      movel([0.335259, -1.470222, -2.504094, -0.738074, 1.570796, 1.906055],accel_mss,speed_ms,0,blend_radius_m)
      movel([0.336291, -1.468662, -2.505402, -0.738325, 1.570796, 1.907087],accel_mss,speed_ms,0,blend_radius_m)
      movel([0.337329, -1.467098, -2.506710, -0.738581, 1.570796, 1.908125],accel_mss,speed_ms,0,blend_radius_m)
      movel([0.339195, -1.464306, -2.509036, -0.739047, 1.570796, 1.909991],accel_mss,speed_ms,0,blend_radius_m)
      movel([0.339233, -1.464257, -2.509076, -0.739055, 1.570796, 1.910029],accel_mss,speed_ms,0,blend_radius_m)
      movel([0.339275, -1.464212, -2.509113, -0.739063, 1.570796, 1.910071],accel_mss,speed_ms,0,blend_radius_m)
      movel([0.339324, -1.464171, -2.509148, -0.739070, 1.570796, 1.910121],accel_mss,speed_ms,0,blend_radius_m)
      movel([0.339395, -1.464123, -2.509187, -0.739078, 1.570796, 1.910192],accel_mss,speed_ms,0,blend_radius_m)
      movel([0.339472, -1.464083, -2.509221, -0.739085, 1.570796, 1.910268],accel_mss,speed_ms,0,blend_radius_m)
      movel([0.339550, -1.464051, -2.509248, -0.739090, 1.570796, 1.910346],accel_mss,speed_ms,0,blend_radius_m)
      movel([0.339628, -1.464028, -2.509266, -0.739094, 1.570796, 1.910425],accel_mss,speed_ms,0,blend_radius_m)
      movel([0.343643, -1.463141, -2.510002, -0.739245, 1.570796, 1.914440],accel_mss,speed_ms,0,blend_radius_m)
      movel([0.345543, -1.462730, -2.510343, -0.739316, 1.570796, 1.916340],accel_mss,speed_ms,0,blend_radius_m)
      movel([0.347442, -1.462325, -2.510678, -0.739385, 1.570796, 1.918239],accel_mss,speed_ms,0,blend_radius_m)
      movel([0.347658, -1.462283, -2.510713, -0.739393, 1.570796, 1.918454],accel_mss,speed_ms,0,blend_radius_m)
      movel([0.347869, -1.462252, -2.510739, -0.739398, 1.570796, 1.918666],accel_mss,speed_ms,0,blend_radius_m)
      movel([0.348080, -1.462228, -2.510759, -0.739402, 1.570796, 1.918876],accel_mss,speed_ms,0,blend_radius_m)
      movel([0.348287, -1.462214, -2.510770, -0.739405, 1.570796, 1.919083],accel_mss,speed_ms,0,blend_radius_m)
      movel([0.348391, -1.462213, -2.510771, -0.739405, 1.570796, 1.919187],accel_mss,speed_ms,0,blend_radius_m)
      movel([0.348491, -1.462224, -2.510762, -0.739403, 1.570796, 1.919287],accel_mss,speed_ms,0,blend_radius_m)
      movel([0.348582, -1.462246, -2.510744, -0.739399, 1.570796, 1.919378],accel_mss,speed_ms,0,blend_radius_m)
      movel([0.348667, -1.462277, -2.510718, -0.739394, 1.570796, 1.919464],accel_mss,speed_ms,0,blend_radius_m)
      movel([0.355079, -1.465147, -2.508336, -0.738906, 1.570796, 1.925875],accel_mss,speed_ms,0,blend_radius_m)
      movel([0.361512, -1.468104, -2.505869, -0.738416, 1.570796, 1.932309],accel_mss,speed_ms,0,blend_radius_m)
      speed_ms = 0.003
      movel([0.361512, -1.456047, -2.500408, -0.755934, 1.570796, 1.932309],accel_mss,speed_ms,0,blend_radius_m)
      speed_ms = 0.01
      movel([0.361512, -1.432785, -2.489096, -0.790508, 1.570796, 1.932309],accel_mss,speed_ms,0,blend_radius_m)
      movel([0.379710, -1.378240, -2.530192, -0.803957, 1.570796, 1.950507],accel_mss,speed_ms,0,blend_radius_m)
      movel([0.379710, -1.402570, -2.542172, -0.767647, 1.570796, 1.950507],accel_mss,speed_ms,0,blend_radius_m)
      speed_ms = 0.003
      movel([0.379710, -1.412031, -2.546529, -0.753828, 1.570796, 1.950507],accel_mss,speed_ms,0,blend_radius_m)
      speed_ms = 0.007
      movel([0.362253, -1.410756, -2.547488, -0.754145, 1.570796, 1.933049],accel_mss,speed_ms,0,blend_radius_m)
      movel([0.344648, -1.409792, -2.548210, -0.754386, 1.570796, 1.915445],accel_mss,speed_ms,0,blend_radius_m)
      movel([0.344585, -1.409783, -2.548217, -0.754389, 1.570796, 1.915381],accel_mss,speed_ms,0,blend_radius_m)
      movel([0.344531, -1.409760, -2.548234, -0.754395, 1.570796, 1.915327],accel_mss,speed_ms,0,blend_radius_m)
      movel([0.344488, -1.409724, -2.548261, -0.754404, 1.570796, 1.915285],accel_mss,speed_ms,0,blend_radius_m)
      movel([0.344479, -1.409701, -2.548278, -0.754409, 1.570796, 1.915276],accel_mss,speed_ms,0,blend_radius_m)
      movel([0.344486, -1.409671, -2.548301, -0.754417, 1.570796, 1.915282],accel_mss,speed_ms,0,blend_radius_m)
      movel([0.345097, -1.408321, -2.549311, -0.754757, 1.570796, 1.915893],accel_mss,speed_ms,0,blend_radius_m)
      movel([0.345789, -1.406806, -2.550440, -0.755143, 1.570796, 1.916585],accel_mss,speed_ms,0,blend_radius_m)
      movel([0.346623, -1.405010, -2.551775, -0.755604, 1.570796, 1.917420],accel_mss,speed_ms,0,blend_radius_m)
      movel([0.348821, -1.400311, -2.555246, -0.756833, 1.570796, 1.919617],accel_mss,speed_ms,0,blend_radius_m)
      movel([0.349537, -1.400351, -2.555216, -0.756822, 1.570796, 1.920333],accel_mss,speed_ms,0,blend_radius_m)
      movel([0.355122, -1.400638, -2.555005, -0.756746, 1.570796, 1.925918],accel_mss,speed_ms,0,blend_radius_m)
      movel([0.367492, -1.401377, -2.554461, -0.756551, 1.570796, 1.938288],accel_mss,speed_ms,0,blend_radius_m)
      movel([0.384563, -1.402661, -2.553514, -0.756214, 1.570796, 1.955359],accel_mss,speed_ms,0,blend_radius_m)
      movel([0.384371, -1.403120, -2.553175, -0.756094, 1.570796, 1.955168],accel_mss,speed_ms,0,blend_radius_m)
      movel([0.384269, -1.403350, -2.553005, -0.756034, 1.570796, 1.955065],accel_mss,speed_ms,0,blend_radius_m)
      movel([0.384107, -1.403677, -2.552763, -0.755949, 1.570796, 1.954904],accel_mss,speed_ms,0,blend_radius_m)
      movel([0.383922, -1.404034, -2.552499, -0.755856, 1.570796, 1.954719],accel_mss,speed_ms,0,blend_radius_m)
      movel([0.383739, -1.404372, -2.552248, -0.755769, 1.570796, 1.954535],accel_mss,speed_ms,0,blend_radius_m)
      movel([0.383297, -1.405163, -2.551661, -0.755564, 1.570796, 1.954093],accel_mss,speed_ms,0,blend_radius_m)
      movel([0.381035, -1.405216, -2.551623, -0.755551, 1.570796, 1.951831],accel_mss,speed_ms,0,blend_radius_m)
      movel([0.378702, -1.405326, -2.551541, -0.755522, 1.570796, 1.949498],accel_mss,speed_ms,0,blend_radius_m)
      movel([0.378649, -1.405401, -2.551485, -0.755503, 1.570796, 1.949445],accel_mss,speed_ms,0,blend_radius_m)
      movel([0.377743, -1.408698, -2.549029, -0.754662, 1.570796, 1.948539],accel_mss,speed_ms,0,blend_radius_m)
      movel([0.381641, -1.408475, -2.549196, -0.754719, 1.570796, 1.952437],accel_mss,speed_ms,0,blend_radius_m)
      movel([0.380797, -1.410194, -2.547909, -0.754286, 1.570796, 1.951594],accel_mss,speed_ms,0,blend_radius_m)
      movel([0.380468, -1.410858, -2.547411, -0.754120, 1.570796, 1.951265],accel_mss,speed_ms,0,blend_radius_m)
      movel([0.380174, -1.411429, -2.546983, -0.753978, 1.570796, 1.950970],accel_mss,speed_ms,0,blend_radius_m)
      movel([0.379918, -1.411918, -2.546614, -0.753856, 1.570796, 1.950714],accel_mss,speed_ms,0,blend_radius_m)
      movel([0.379892, -1.411953, -2.546588, -0.753848, 1.570796, 1.950688],accel_mss,speed_ms,0,blend_radius_m)
      movel([0.379860, -1.411982, -2.546567, -0.753841, 1.570796, 1.950656],accel_mss,speed_ms,0,blend_radius_m)
      movel([0.379809, -1.412013, -2.546544, -0.753833, 1.570796, 1.950606],accel_mss,speed_ms,0,blend_radius_m)
      movel([0.379758, -1.412028, -2.546532, -0.753829, 1.570796, 1.950555],accel_mss,speed_ms,0,blend_radius_m)
      movel([0.379710, -1.412031, -2.546529, -0.753828, 1.570796, 1.950507],accel_mss,speed_ms,0,blend_radius_m)
      speed_ms = 0.003
      movel([0.379710, -1.415226, -2.547965, -0.749197, 1.570796, 1.950507],accel_mss,speed_ms,0,blend_radius_m)
      speed_ms = 0.007
      movel([0.362253, -1.413954, -2.548926, -0.749509, 1.570796, 1.933049],accel_mss,speed_ms,0,blend_radius_m)
      movel([0.344648, -1.412994, -2.549649, -0.749746, 1.570796, 1.915445],accel_mss,speed_ms,0,blend_radius_m)
      movel([0.344585, -1.412984, -2.549657, -0.749748, 1.570796, 1.915381],accel_mss,speed_ms,0,blend_radius_m)
      movel([0.344531, -1.412962, -2.549674, -0.749754, 1.570796, 1.915327],accel_mss,speed_ms,0,blend_radius_m)
      movel([0.344488, -1.412926, -2.549701, -0.749763, 1.570796, 1.915285],accel_mss,speed_ms,0,blend_radius_m)
      movel([0.344479, -1.412903, -2.549718, -0.749768, 1.570796, 1.915276],accel_mss,speed_ms,0,blend_radius_m)
      movel([0.344486, -1.412873, -2.549740, -0.749776, 1.570796, 1.915282],accel_mss,speed_ms,0,blend_radius_m)
      movel([0.345097, -1.411526, -2.550752, -0.750110, 1.570796, 1.915893],accel_mss,speed_ms,0,blend_radius_m)
      movel([0.345789, -1.410016, -2.551885, -0.750489, 1.570796, 1.916585],accel_mss,speed_ms,0,blend_radius_m)
      movel([0.346623, -1.408225, -2.553222, -0.750942, 1.570796, 1.917420],accel_mss,speed_ms,0,blend_radius_m)
      movel([0.348821, -1.403539, -2.556700, -0.752150, 1.570796, 1.919617],accel_mss,speed_ms,0,blend_radius_m)
      movel([0.349537, -1.403579, -2.556670, -0.752139, 1.570796, 1.920333],accel_mss,speed_ms,0,blend_radius_m)
      movel([0.355122, -1.403865, -2.556459, -0.752065, 1.570796, 1.925918],accel_mss,speed_ms,0,blend_radius_m)
      movel([0.367492, -1.404602, -2.555914, -0.751873, 1.570796, 1.938288],accel_mss,speed_ms,0,blend_radius_m)
      movel([0.384563, -1.405883, -2.554965, -0.751542, 1.570796, 1.955359],accel_mss,speed_ms,0,blend_radius_m)
      movel([0.384371, -1.406340, -2.554625, -0.751424, 1.570796, 1.955168],accel_mss,speed_ms,0,blend_radius_m)
      movel([0.384269, -1.406569, -2.554455, -0.751365, 1.570796, 1.955065],accel_mss,speed_ms,0,blend_radius_m)
      movel([0.384107, -1.406895, -2.554212, -0.751281, 1.570796, 1.954904],accel_mss,speed_ms,0,blend_radius_m)
      movel([0.383922, -1.407252, -2.553947, -0.751190, 1.570796, 1.954719],accel_mss,speed_ms,0,blend_radius_m)
      movel([0.383739, -1.407589, -2.553696, -0.751104, 1.570796, 1.954535],accel_mss,speed_ms,0,blend_radius_m)
      movel([0.383297, -1.408378, -2.553108, -0.750903, 1.570796, 1.954093],accel_mss,speed_ms,0,blend_radius_m)
      movel([0.381035, -1.408430, -2.553069, -0.750890, 1.570796, 1.951831],accel_mss,speed_ms,0,blend_radius_m)
      movel([0.378702, -1.408540, -2.552987, -0.750862, 1.570796, 1.949498],accel_mss,speed_ms,0,blend_radius_m)
      movel([0.378649, -1.408615, -2.552931, -0.750843, 1.570796, 1.949445],accel_mss,speed_ms,0,blend_radius_m)
      movel([0.377743, -1.411903, -2.550470, -0.750016, 1.570796, 1.948539],accel_mss,speed_ms,0,blend_radius_m)
      movel([0.381641, -1.411680, -2.550637, -0.750072, 1.570796, 1.952437],accel_mss,speed_ms,0,blend_radius_m)
      movel([0.380797, -1.413394, -2.549348, -0.749647, 1.570796, 1.951594],accel_mss,speed_ms,0,blend_radius_m)
      movel([0.380468, -1.414056, -2.548849, -0.749484, 1.570796, 1.951265],accel_mss,speed_ms,0,blend_radius_m)
      movel([0.380174, -1.414625, -2.548419, -0.749344, 1.570796, 1.950970],accel_mss,speed_ms,0,blend_radius_m)
      movel([0.379918, -1.415114, -2.548050, -0.749225, 1.570796, 1.950714],accel_mss,speed_ms,0,blend_radius_m)
      movel([0.379892, -1.415148, -2.548024, -0.749217, 1.570796, 1.950688],accel_mss,speed_ms,0,blend_radius_m)
      movel([0.379860, -1.415177, -2.548003, -0.749210, 1.570796, 1.950656],accel_mss,speed_ms,0,blend_radius_m)
      movel([0.379809, -1.415208, -2.547979, -0.749202, 1.570796, 1.950606],accel_mss,speed_ms,0,blend_radius_m)
      movel([0.379758, -1.415223, -2.547967, -0.749198, 1.570796, 1.950555],accel_mss,speed_ms,0,blend_radius_m)
      movel([0.379710, -1.415226, -2.547965, -0.749197, 1.570796, 1.950507],accel_mss,speed_ms,0,blend_radius_m)
      speed_ms = 0.003
      movel([0.379710, -1.402570, -2.542172, -0.767647, 1.570796, 1.950507],accel_mss,speed_ms,0,blend_radius_m)
      speed_ms = 0.01
      movel([0.379710, -1.378240, -2.530192, -0.803957, 1.570796, 1.950507],accel_mss,speed_ms,0,blend_radius_m)
      movel([0.382022, -1.366015, -2.538831, -0.807543, 1.570796, 1.952818],accel_mss,speed_ms,0,blend_radius_m)
      movel([0.382022, -1.390572, -2.550964, -0.770853, 1.570796, 1.952818],accel_mss,speed_ms,0,blend_radius_m)
      speed_ms = 0.003
      movel([0.382022, -1.400129, -2.555379, -0.756881, 1.570796, 1.952818],accel_mss,speed_ms,0,blend_radius_m)
      speed_ms = 0.007
      movel([0.381906, -1.400143, -2.555369, -0.756877, 1.570796, 1.952702],accel_mss,speed_ms,0,blend_radius_m)
      movel([0.381797, -1.400145, -2.555368, -0.756877, 1.570796, 1.952593],accel_mss,speed_ms,0,blend_radius_m)
      movel([0.381615, -1.400131, -2.555378, -0.756880, 1.570796, 1.952411],accel_mss,speed_ms,0,blend_radius_m)
      movel([0.381436, -1.400113, -2.555391, -0.756885, 1.570796, 1.952232],accel_mss,speed_ms,0,blend_radius_m)
      movel([0.380003, -1.399974, -2.555493, -0.756922, 1.570796, 1.950799],accel_mss,speed_ms,0,blend_radius_m)
      movel([0.365041, -1.398928, -2.556261, -0.757200, 1.570796, 1.935837],accel_mss,speed_ms,0,blend_radius_m)
      movel([0.349510, -1.398092, -2.556873, -0.757424, 1.570796, 1.920307],accel_mss,speed_ms,0,blend_radius_m)
      movel([0.348976, -1.398094, -2.556871, -0.757423, 1.570796, 1.919772],accel_mss,speed_ms,0,blend_radius_m)
      movel([0.348929, -1.398092, -2.556873, -0.757424, 1.570796, 1.919725],accel_mss,speed_ms,0,blend_radius_m)
      movel([0.348886, -1.398079, -2.556882, -0.757427, 1.570796, 1.919683],accel_mss,speed_ms,0,blend_radius_m)
      movel([0.348854, -1.398057, -2.556898, -0.757433, 1.570796, 1.919650],accel_mss,speed_ms,0,blend_radius_m)
      movel([0.348827, -1.398026, -2.556921, -0.757442, 1.570796, 1.919624],accel_mss,speed_ms,0,blend_radius_m)
      movel([0.348812, -1.397990, -2.556947, -0.757451, 1.570796, 1.919608],accel_mss,speed_ms,0,blend_radius_m)
      movel([0.348808, -1.397947, -2.556979, -0.757463, 1.570796, 1.919604],accel_mss,speed_ms,0,blend_radius_m)
      movel([0.348816, -1.397841, -2.557057, -0.757491, 1.570796, 1.919613],accel_mss,speed_ms,0,blend_radius_m)
      movel([0.348845, -1.397731, -2.557137, -0.757521, 1.570796, 1.919641],accel_mss,speed_ms,0,blend_radius_m)
      movel([0.348908, -1.397546, -2.557272, -0.757571, 1.570796, 1.919705],accel_mss,speed_ms,0,blend_radius_m)
      movel([0.348977, -1.397359, -2.557409, -0.757621, 1.570796, 1.919774],accel_mss,speed_ms,0,blend_radius_m)
      movel([0.349097, -1.397073, -2.557618, -0.757698, 1.570796, 1.919894],accel_mss,speed_ms,0,blend_radius_m)
      movel([0.349227, -1.396787, -2.557827, -0.757775, 1.570796, 1.920023],accel_mss,speed_ms,0,blend_radius_m)
      movel([0.351083, -1.392872, -2.560673, -0.758844, 1.570796, 1.921879],accel_mss,speed_ms,0,blend_radius_m)
      movel([0.353252, -1.388325, -2.563951, -0.760113, 1.570796, 1.924049],accel_mss,speed_ms,0,blend_radius_m)
      movel([0.355797, -1.383031, -2.567730, -0.761628, 1.570796, 1.926593],accel_mss,speed_ms,0,blend_radius_m)
      movel([0.362519, -1.369156, -2.577443, -0.765790, 1.570796, 1.933315],accel_mss,speed_ms,0,blend_radius_m)
      movel([0.363532, -1.369162, -2.577439, -0.765788, 1.570796, 1.934328],accel_mss,speed_ms,0,blend_radius_m)
      movel([0.364039, -1.369170, -2.577434, -0.765786, 1.570796, 1.934835],accel_mss,speed_ms,0,blend_radius_m)
      movel([0.364541, -1.369192, -2.577419, -0.765779, 1.570796, 1.935337],accel_mss,speed_ms,0,blend_radius_m)
      movel([0.365033, -1.369226, -2.577395, -0.765768, 1.570796, 1.935829],accel_mss,speed_ms,0,blend_radius_m)
      movel([0.365522, -1.369271, -2.577364, -0.765754, 1.570796, 1.936319],accel_mss,speed_ms,0,blend_radius_m)
      movel([0.366251, -1.369359, -2.577303, -0.765727, 1.570796, 1.937047],accel_mss,speed_ms,0,blend_radius_m)
      movel([0.366968, -1.369467, -2.577228, -0.765694, 1.570796, 1.937764],accel_mss,speed_ms,0,blend_radius_m)
      movel([0.367676, -1.369589, -2.577144, -0.765656, 1.570796, 1.938472],accel_mss,speed_ms,0,blend_radius_m)
      movel([0.368391, -1.369734, -2.577044, -0.765611, 1.570796, 1.939187],accel_mss,speed_ms,0,blend_radius_m)
      movel([0.369092, -1.369897, -2.576932, -0.765561, 1.570796, 1.939888],accel_mss,speed_ms,0,blend_radius_m)
      movel([0.369784, -1.370076, -2.576808, -0.765506, 1.570796, 1.940580],accel_mss,speed_ms,0,blend_radius_m)
      movel([0.370258, -1.370210, -2.576715, -0.765464, 1.570796, 1.941054],accel_mss,speed_ms,0,blend_radius_m)
      movel([0.370723, -1.370357, -2.576613, -0.765419, 1.570796, 1.941519],accel_mss,speed_ms,0,blend_radius_m)
      movel([0.371180, -1.370516, -2.576503, -0.765370, 1.570796, 1.941977],accel_mss,speed_ms,0,blend_radius_m)
      movel([0.371629, -1.370684, -2.576387, -0.765318, 1.570796, 1.942425],accel_mss,speed_ms,0,blend_radius_m)
      movel([0.372272, -1.370949, -2.576203, -0.765237, 1.570796, 1.943068],accel_mss,speed_ms,0,blend_radius_m)
      movel([0.372898, -1.371228, -2.576010, -0.765151, 1.570796, 1.943695],accel_mss,speed_ms,0,blend_radius_m)
      movel([0.373510, -1.371527, -2.575803, -0.765059, 1.570796, 1.944307],accel_mss,speed_ms,0,blend_radius_m)
      movel([0.374110, -1.371842, -2.575584, -0.764963, 1.570796, 1.944907],accel_mss,speed_ms,0,blend_radius_m)
      movel([0.374692, -1.372172, -2.575355, -0.764862, 1.570796, 1.945489],accel_mss,speed_ms,0,blend_radius_m)
      movel([0.375259, -1.372520, -2.575113, -0.764756, 1.570796, 1.946055],accel_mss,speed_ms,0,blend_radius_m)
      movel([0.375812, -1.372886, -2.574859, -0.764644, 1.570796, 1.946608],accel_mss,speed_ms,0,blend_radius_m)
      movel([0.376347, -1.373266, -2.574595, -0.764529, 1.570796, 1.947143],accel_mss,speed_ms,0,blend_radius_m)
      movel([0.376865, -1.373662, -2.574318, -0.764408, 1.570796, 1.947661],accel_mss,speed_ms,0,blend_radius_m)
      movel([0.377367, -1.374074, -2.574032, -0.764283, 1.570796, 1.948164],accel_mss,speed_ms,0,blend_radius_m)
      movel([0.377848, -1.374497, -2.573737, -0.764155, 1.570796, 1.948645],accel_mss,speed_ms,0,blend_radius_m)
      movel([0.378310, -1.374937, -2.573430, -0.764023, 1.570796, 1.949107],accel_mss,speed_ms,0,blend_radius_m)
      movel([0.378755, -1.375391, -2.573112, -0.763886, 1.570796, 1.949551],accel_mss,speed_ms,0,blend_radius_m)
      movel([0.379183, -1.375859, -2.572785, -0.763745, 1.570796, 1.949979],accel_mss,speed_ms,0,blend_radius_m)
      movel([0.379591, -1.376342, -2.572447, -0.763600, 1.570796, 1.950388],accel_mss,speed_ms,0,blend_radius_m)
      movel([0.379981, -1.376840, -2.572098, -0.763451, 1.570796, 1.950777],accel_mss,speed_ms,0,blend_radius_m)
      movel([0.380354, -1.377351, -2.571739, -0.763298, 1.570796, 1.951150],accel_mss,speed_ms,0,blend_radius_m)
      movel([0.380706, -1.377876, -2.571371, -0.763142, 1.570796, 1.951502],accel_mss,speed_ms,0,blend_radius_m)
      movel([0.381041, -1.378415, -2.570992, -0.762982, 1.570796, 1.951837],accel_mss,speed_ms,0,blend_radius_m)
      movel([0.381356, -1.378965, -2.570605, -0.762819, 1.570796, 1.952153],accel_mss,speed_ms,0,blend_radius_m)
      movel([0.381656, -1.379536, -2.570203, -0.762651, 1.570796, 1.952452],accel_mss,speed_ms,0,blend_radius_m)
      movel([0.381939, -1.380118, -2.569792, -0.762479, 1.570796, 1.952735],accel_mss,speed_ms,0,blend_radius_m)
      movel([0.382200, -1.380714, -2.569371, -0.762304, 1.570796, 1.952996],accel_mss,speed_ms,0,blend_radius_m)
      movel([0.382442, -1.381320, -2.568943, -0.762126, 1.570796, 1.953238],accel_mss,speed_ms,0,blend_radius_m)
      movel([0.382666, -1.381936, -2.568506, -0.761946, 1.570796, 1.953462],accel_mss,speed_ms,0,blend_radius_m)
      movel([0.382868, -1.382564, -2.568061, -0.761764, 1.570796, 1.953664],accel_mss,speed_ms,0,blend_radius_m)
      movel([0.383052, -1.383202, -2.567609, -0.761579, 1.570796, 1.953848],accel_mss,speed_ms,0,blend_radius_m)
      movel([0.383215, -1.383850, -2.567148, -0.761391, 1.570796, 1.954011],accel_mss,speed_ms,0,blend_radius_m)
      movel([0.383358, -1.384508, -2.566680, -0.761201, 1.570796, 1.954154],accel_mss,speed_ms,0,blend_radius_m)
      movel([0.383483, -1.385174, -2.566205, -0.761010, 1.570796, 1.954279],accel_mss,speed_ms,0,blend_radius_m)
      movel([0.383590, -1.385871, -2.565708, -0.760810, 1.570796, 1.954386],accel_mss,speed_ms,0,blend_radius_m)
      movel([0.383679, -1.386577, -2.565203, -0.760609, 1.570796, 1.954475],accel_mss,speed_ms,0,blend_radius_m)
      movel([0.383752, -1.387290, -2.564693, -0.760406, 1.570796, 1.954548],accel_mss,speed_ms,0,blend_radius_m)
      movel([0.383803, -1.388009, -2.564178, -0.760202, 1.570796, 1.954599],accel_mss,speed_ms,0,blend_radius_m)
      movel([0.383837, -1.388735, -2.563657, -0.759997, 1.570796, 1.954633],accel_mss,speed_ms,0,blend_radius_m)
      movel([0.383854, -1.389469, -2.563129, -0.759791, 1.570796, 1.954650],accel_mss,speed_ms,0,blend_radius_m)
      movel([0.383851, -1.390207, -2.562598, -0.759584, 1.570796, 1.954647],accel_mss,speed_ms,0,blend_radius_m)
      movel([0.383828, -1.390952, -2.562061, -0.759376, 1.570796, 1.954625],accel_mss,speed_ms,0,blend_radius_m)
      movel([0.383790, -1.391700, -2.561521, -0.759168, 1.570796, 1.954587],accel_mss,speed_ms,0,blend_radius_m)
      movel([0.383731, -1.392455, -2.560975, -0.758959, 1.570796, 1.954528],accel_mss,speed_ms,0,blend_radius_m)
      movel([0.383683, -1.392933, -2.560629, -0.758827, 1.570796, 1.954479],accel_mss,speed_ms,0,blend_radius_m)
      movel([0.383624, -1.393413, -2.560281, -0.758695, 1.570796, 1.954421],accel_mss,speed_ms,0,blend_radius_m)
      movel([0.383552, -1.393897, -2.559930, -0.758562, 1.570796, 1.954349],accel_mss,speed_ms,0,blend_radius_m)
      movel([0.383390, -1.394883, -2.559214, -0.758292, 1.570796, 1.954186],accel_mss,speed_ms,0,blend_radius_m)
      movel([0.383211, -1.395870, -2.558495, -0.758024, 1.570796, 1.954008],accel_mss,speed_ms,0,blend_radius_m)
      movel([0.383022, -1.396842, -2.557786, -0.757760, 1.570796, 1.953819],accel_mss,speed_ms,0,blend_radius_m)
      movel([0.382822, -1.397816, -2.557075, -0.757498, 1.570796, 1.953618],accel_mss,speed_ms,0,blend_radius_m)
      movel([0.382723, -1.398249, -2.556758, -0.757382, 1.570796, 1.953519],accel_mss,speed_ms,0,blend_radius_m)
      movel([0.382610, -1.398685, -2.556439, -0.757265, 1.570796, 1.953406],accel_mss,speed_ms,0,blend_radius_m)
      movel([0.382485, -1.399121, -2.556119, -0.757149, 1.570796, 1.953281],accel_mss,speed_ms,0,blend_radius_m)
      movel([0.382217, -1.400005, -2.555470, -0.756914, 1.570796, 1.953014],accel_mss,speed_ms,0,blend_radius_m)
      movel([0.382192, -1.400038, -2.555446, -0.756905, 1.570796, 1.952989],accel_mss,speed_ms,0,blend_radius_m)
      movel([0.382157, -1.400070, -2.555423, -0.756896, 1.570796, 1.952953],accel_mss,speed_ms,0,blend_radius_m)
      movel([0.382114, -1.400097, -2.555403, -0.756889, 1.570796, 1.952910],accel_mss,speed_ms,0,blend_radius_m)
      movel([0.382067, -1.400117, -2.555388, -0.756884, 1.570796, 1.952864],accel_mss,speed_ms,0,blend_radius_m)
      movel([0.382022, -1.400129, -2.555379, -0.756881, 1.570796, 1.952818],accel_mss,speed_ms,0,blend_radius_m)
      speed_ms = 0.003
      movel([0.382022, -1.403358, -2.556834, -0.752197, 1.570796, 1.952818],accel_mss,speed_ms,0,blend_radius_m)
      speed_ms = 0.007
      movel([0.381906, -1.403371, -2.556824, -0.752194, 1.570796, 1.952702],accel_mss,speed_ms,0,blend_radius_m)
      movel([0.381797, -1.403373, -2.556823, -0.752193, 1.570796, 1.952593],accel_mss,speed_ms,0,blend_radius_m)
      movel([0.381615, -1.403360, -2.556833, -0.752197, 1.570796, 1.952411],accel_mss,speed_ms,0,blend_radius_m)
      movel([0.381436, -1.403342, -2.556846, -0.752202, 1.570796, 1.952232],accel_mss,speed_ms,0,blend_radius_m)
      movel([0.380003, -1.403203, -2.556948, -0.752238, 1.570796, 1.950799],accel_mss,speed_ms,0,blend_radius_m)
      movel([0.365041, -1.402159, -2.557718, -0.752512, 1.570796, 1.935837],accel_mss,speed_ms,0,blend_radius_m)
      movel([0.349510, -1.401326, -2.558331, -0.752732, 1.570796, 1.920307],accel_mss,speed_ms,0,blend_radius_m)
      movel([0.348976, -1.401328, -2.558330, -0.752731, 1.570796, 1.919772],accel_mss,speed_ms,0,blend_radius_m)
      movel([0.348929, -1.401326, -2.558331, -0.752732, 1.570796, 1.919725],accel_mss,speed_ms,0,blend_radius_m)
      movel([0.348886, -1.401314, -2.558340, -0.752735, 1.570796, 1.919683],accel_mss,speed_ms,0,blend_radius_m)
      movel([0.348854, -1.401291, -2.558357, -0.752741, 1.570796, 1.919650],accel_mss,speed_ms,0,blend_radius_m)
      movel([0.348827, -1.401261, -2.558379, -0.752749, 1.570796, 1.919624],accel_mss,speed_ms,0,blend_radius_m)
      movel([0.348812, -1.401225, -2.558406, -0.752759, 1.570796, 1.919608],accel_mss,speed_ms,0,blend_radius_m)
      movel([0.348808, -1.401182, -2.558437, -0.752770, 1.570796, 1.919604],accel_mss,speed_ms,0,blend_radius_m)
      movel([0.348816, -1.401076, -2.558515, -0.752798, 1.570796, 1.919613],accel_mss,speed_ms,0,blend_radius_m)
      movel([0.348845, -1.400966, -2.558596, -0.752827, 1.570796, 1.919641],accel_mss,speed_ms,0,blend_radius_m)
      movel([0.348908, -1.400782, -2.558731, -0.752876, 1.570796, 1.919705],accel_mss,speed_ms,0,blend_radius_m)
      movel([0.348977, -1.400595, -2.558869, -0.752926, 1.570796, 1.919774],accel_mss,speed_ms,0,blend_radius_m)
      movel([0.349097, -1.400310, -2.559078, -0.753001, 1.570796, 1.919894],accel_mss,speed_ms,0,blend_radius_m)
      movel([0.349227, -1.400024, -2.559287, -0.753077, 1.570796, 1.920023],accel_mss,speed_ms,0,blend_radius_m)
      movel([0.351083, -1.396121, -2.562140, -0.754129, 1.570796, 1.921879],accel_mss,speed_ms,0,blend_radius_m)
      movel([0.353252, -1.391586, -2.565425, -0.755378, 1.570796, 1.924049],accel_mss,speed_ms,0,blend_radius_m)
      movel([0.355797, -1.386307, -2.569212, -0.756870, 1.570796, 1.926593],accel_mss,speed_ms,0,blend_radius_m)
      movel([0.362519, -1.372469, -2.578948, -0.760972, 1.570796, 1.933315],accel_mss,speed_ms,0,blend_radius_m)
      movel([0.363532, -1.372475, -2.578944, -0.760970, 1.570796, 1.934328],accel_mss,speed_ms,0,blend_radius_m)
      movel([0.364039, -1.372482, -2.578939, -0.760968, 1.570796, 1.934835],accel_mss,speed_ms,0,blend_radius_m)
      movel([0.364541, -1.372504, -2.578924, -0.760961, 1.570796, 1.935337],accel_mss,speed_ms,0,blend_radius_m)
      movel([0.365033, -1.372538, -2.578900, -0.760951, 1.570796, 1.935829],accel_mss,speed_ms,0,blend_radius_m)
      movel([0.365522, -1.372583, -2.578869, -0.760937, 1.570796, 1.936319],accel_mss,speed_ms,0,blend_radius_m)
      movel([0.366251, -1.372672, -2.578808, -0.760910, 1.570796, 1.937047],accel_mss,speed_ms,0,blend_radius_m)
      movel([0.366968, -1.372779, -2.578733, -0.760877, 1.570796, 1.937764],accel_mss,speed_ms,0,blend_radius_m)
      movel([0.367676, -1.372901, -2.578649, -0.760840, 1.570796, 1.938472],accel_mss,speed_ms,0,blend_radius_m)
      movel([0.368391, -1.373045, -2.578548, -0.760795, 1.570796, 1.939187],accel_mss,speed_ms,0,blend_radius_m)
      movel([0.369092, -1.373207, -2.578436, -0.760746, 1.570796, 1.939888],accel_mss,speed_ms,0,blend_radius_m)
      movel([0.369784, -1.373386, -2.578312, -0.760691, 1.570796, 1.940580],accel_mss,speed_ms,0,blend_radius_m)
      movel([0.370258, -1.373520, -2.578218, -0.760650, 1.570796, 1.941054],accel_mss,speed_ms,0,blend_radius_m)
      movel([0.370723, -1.373667, -2.578116, -0.760606, 1.570796, 1.941519],accel_mss,speed_ms,0,blend_radius_m)
      movel([0.371180, -1.373825, -2.578006, -0.760558, 1.570796, 1.941977],accel_mss,speed_ms,0,blend_radius_m)
      movel([0.371629, -1.373993, -2.577890, -0.760507, 1.570796, 1.942425],accel_mss,speed_ms,0,blend_radius_m)
      movel([0.372272, -1.374257, -2.577706, -0.760426, 1.570796, 1.943068],accel_mss,speed_ms,0,blend_radius_m)
      movel([0.372898, -1.374535, -2.577512, -0.760342, 1.570796, 1.943695],accel_mss,speed_ms,0,blend_radius_m)
      movel([0.373510, -1.374833, -2.577305, -0.760252, 1.570796, 1.944307],accel_mss,speed_ms,0,blend_radius_m)
      movel([0.374110, -1.375147, -2.577085, -0.760156, 1.570796, 1.944907],accel_mss,speed_ms,0,blend_radius_m)
      movel([0.374692, -1.375476, -2.576856, -0.760057, 1.570796, 1.945489],accel_mss,speed_ms,0,blend_radius_m)
      movel([0.375259, -1.375824, -2.576613, -0.759952, 1.570796, 1.946055],accel_mss,speed_ms,0,blend_radius_m)
      movel([0.375812, -1.376188, -2.576358, -0.759842, 1.570796, 1.946608],accel_mss,speed_ms,0,blend_radius_m)
      movel([0.376347, -1.376567, -2.576093, -0.759728, 1.570796, 1.947143],accel_mss,speed_ms,0,blend_radius_m)
      movel([0.376865, -1.376963, -2.575817, -0.759609, 1.570796, 1.947661],accel_mss,speed_ms,0,blend_radius_m)
      movel([0.377367, -1.377373, -2.575529, -0.759487, 1.570796, 1.948164],accel_mss,speed_ms,0,blend_radius_m)
      movel([0.377848, -1.377795, -2.575233, -0.759360, 1.570796, 1.948645],accel_mss,speed_ms,0,blend_radius_m)
      movel([0.378310, -1.378234, -2.574926, -0.759229, 1.570796, 1.949107],accel_mss,speed_ms,0,blend_radius_m)
      movel([0.378755, -1.378687, -2.574608, -0.759095, 1.570796, 1.949551],accel_mss,speed_ms,0,blend_radius_m)
      movel([0.379183, -1.379154, -2.574279, -0.758956, 1.570796, 1.949979],accel_mss,speed_ms,0,blend_radius_m)
      movel([0.379591, -1.379635, -2.573941, -0.758813, 1.570796, 1.950388],accel_mss,speed_ms,0,blend_radius_m)
      movel([0.379981, -1.380133, -2.573590, -0.758666, 1.570796, 1.950777],accel_mss,speed_ms,0,blend_radius_m)
      movel([0.380354, -1.380642, -2.573231, -0.758516, 1.570796, 1.951150],accel_mss,speed_ms,0,blend_radius_m)
      movel([0.380706, -1.381165, -2.572862, -0.758362, 1.570796, 1.951502],accel_mss,speed_ms,0,blend_radius_m)
      movel([0.381041, -1.381702, -2.572482, -0.758204, 1.570796, 1.951837],accel_mss,speed_ms,0,blend_radius_m)
      movel([0.381356, -1.382251, -2.572094, -0.758043, 1.570796, 1.952153],accel_mss,speed_ms,0,blend_radius_m)
      movel([0.381656, -1.382821, -2.571691, -0.757877, 1.570796, 1.952452],accel_mss,speed_ms,0,blend_radius_m)
      movel([0.381939, -1.383401, -2.571279, -0.757708, 1.570796, 1.952735],accel_mss,speed_ms,0,blend_radius_m)
      movel([0.382200, -1.383996, -2.570857, -0.757536, 1.570796, 1.952996],accel_mss,speed_ms,0,blend_radius_m)
      movel([0.382442, -1.384600, -2.570428, -0.757361, 1.570796, 1.953238],accel_mss,speed_ms,0,blend_radius_m)
      movel([0.382666, -1.385215, -2.569991, -0.757184, 1.570796, 1.953462],accel_mss,speed_ms,0,blend_radius_m)
      movel([0.382868, -1.385841, -2.569544, -0.757003, 1.570796, 1.953664],accel_mss,speed_ms,0,blend_radius_m)
      movel([0.383052, -1.386476, -2.569091, -0.756821, 1.570796, 1.953848],accel_mss,speed_ms,0,blend_radius_m)
      movel([0.383215, -1.387123, -2.568629, -0.756636, 1.570796, 1.954011],accel_mss,speed_ms,0,blend_radius_m)
      movel([0.383358, -1.387779, -2.568160, -0.756450, 1.570796, 1.954154],accel_mss,speed_ms,0,blend_radius_m)
      movel([0.383483, -1.388443, -2.567684, -0.756261, 1.570796, 1.954279],accel_mss,speed_ms,0,blend_radius_m)
      movel([0.383590, -1.389139, -2.567186, -0.756064, 1.570796, 1.954386],accel_mss,speed_ms,0,blend_radius_m)
      movel([0.383679, -1.389843, -2.566680, -0.755866, 1.570796, 1.954475],accel_mss,speed_ms,0,blend_radius_m)
      movel([0.383752, -1.390554, -2.566169, -0.755666, 1.570796, 1.954548],accel_mss,speed_ms,0,blend_radius_m)
      movel([0.383803, -1.391271, -2.565652, -0.755466, 1.570796, 1.954599],accel_mss,speed_ms,0,blend_radius_m)
      movel([0.383837, -1.391995, -2.565130, -0.755264, 1.570796, 1.954633],accel_mss,speed_ms,0,blend_radius_m)
      movel([0.383854, -1.392727, -2.564602, -0.755061, 1.570796, 1.954650],accel_mss,speed_ms,0,blend_radius_m)
      movel([0.383851, -1.393463, -2.564069, -0.754857, 1.570796, 1.954647],accel_mss,speed_ms,0,blend_radius_m)
      movel([0.383828, -1.394205, -2.563531, -0.754653, 1.570796, 1.954625],accel_mss,speed_ms,0,blend_radius_m)
      movel([0.383790, -1.394952, -2.562989, -0.754448, 1.570796, 1.954587],accel_mss,speed_ms,0,blend_radius_m)
      movel([0.383731, -1.395705, -2.562442, -0.754242, 1.570796, 1.954528],accel_mss,speed_ms,0,blend_radius_m)
      movel([0.383683, -1.396181, -2.562096, -0.754112, 1.570796, 1.954479],accel_mss,speed_ms,0,blend_radius_m)
      movel([0.383624, -1.396660, -2.561747, -0.753982, 1.570796, 1.954421],accel_mss,speed_ms,0,blend_radius_m)
      movel([0.383552, -1.397143, -2.561395, -0.753851, 1.570796, 1.954349],accel_mss,speed_ms,0,blend_radius_m)
      movel([0.383390, -1.398126, -2.560677, -0.753586, 1.570796, 1.954186],accel_mss,speed_ms,0,blend_radius_m)
      movel([0.383211, -1.399110, -2.559957, -0.753322, 1.570796, 1.954008],accel_mss,speed_ms,0,blend_radius_m)
      movel([0.383022, -1.400080, -2.559247, -0.753063, 1.570796, 1.953819],accel_mss,speed_ms,0,blend_radius_m)
      movel([0.382822, -1.401051, -2.558534, -0.752805, 1.570796, 1.953618],accel_mss,speed_ms,0,blend_radius_m)
      movel([0.382723, -1.401483, -2.558216, -0.752690, 1.570796, 1.953519],accel_mss,speed_ms,0,blend_radius_m)
      movel([0.382610, -1.401918, -2.557896, -0.752575, 1.570796, 1.953406],accel_mss,speed_ms,0,blend_radius_m)
      movel([0.382485, -1.402352, -2.557576, -0.752461, 1.570796, 1.953281],accel_mss,speed_ms,0,blend_radius_m)
      movel([0.382217, -1.403234, -2.556925, -0.752230, 1.570796, 1.953014],accel_mss,speed_ms,0,blend_radius_m)
      movel([0.382192, -1.403267, -2.556901, -0.752221, 1.570796, 1.952989],accel_mss,speed_ms,0,blend_radius_m)
      movel([0.382157, -1.403298, -2.556878, -0.752213, 1.570796, 1.952953],accel_mss,speed_ms,0,blend_radius_m)
      movel([0.382114, -1.403325, -2.556858, -0.752206, 1.570796, 1.952910],accel_mss,speed_ms,0,blend_radius_m)
      movel([0.382067, -1.403346, -2.556843, -0.752200, 1.570796, 1.952864],accel_mss,speed_ms,0,blend_radius_m)
      movel([0.382022, -1.403358, -2.556834, -0.752197, 1.570796, 1.952818],accel_mss,speed_ms,0,blend_radius_m)
      speed_ms = 0.003
      movel([0.382022, -1.390572, -2.550964, -0.770853, 1.570796, 1.952818],accel_mss,speed_ms,0,blend_radius_m)
      speed_ms = 0.01
      movel([0.382022, -1.366015, -2.538831, -0.807543, 1.570796, 1.952818],accel_mss,speed_ms,0,blend_radius_m)
      movel([0.375158, -1.380220, -2.528774, -0.803396, 1.570796, 1.945954],accel_mss,speed_ms,0,blend_radius_m)
      movel([0.375158, -1.404512, -2.540729, -0.767148, 1.570796, 1.945954],accel_mss,speed_ms,0,blend_radius_m)
      speed_ms = 0.003
      movel([0.375158, -1.413958, -2.545077, -0.753354, 1.570796, 1.945954],accel_mss,speed_ms,0,blend_radius_m)
      speed_ms = 0.007
      movel([0.375180, -1.413964, -2.545073, -0.753352, 1.570796, 1.945976],accel_mss,speed_ms,0,blend_radius_m)
      movel([0.375195, -1.413974, -2.545065, -0.753350, 1.570796, 1.945992],accel_mss,speed_ms,0,blend_radius_m)
      movel([0.375198, -1.413995, -2.545049, -0.753345, 1.570796, 1.945994],accel_mss,speed_ms,0,blend_radius_m)
      movel([0.375187, -1.414017, -2.545033, -0.753339, 1.570796, 1.945983],accel_mss,speed_ms,0,blend_radius_m)
      movel([0.374177, -1.415376, -2.544005, -0.753008, 1.570796, 1.944973],accel_mss,speed_ms,0,blend_radius_m)
      movel([0.373704, -1.416009, -2.543525, -0.752855, 1.570796, 1.944500],accel_mss,speed_ms,0,blend_radius_m)
      movel([0.373225, -1.416638, -2.543048, -0.752703, 1.570796, 1.944021],accel_mss,speed_ms,0,blend_radius_m)
      movel([0.372848, -1.417127, -2.542676, -0.752585, 1.570796, 1.943644],accel_mss,speed_ms,0,blend_radius_m)
      movel([0.372466, -1.417610, -2.542310, -0.752470, 1.570796, 1.943262],accel_mss,speed_ms,0,blend_radius_m)
      movel([0.371969, -1.418221, -2.541844, -0.752324, 1.570796, 1.942765],accel_mss,speed_ms,0,blend_radius_m)
      movel([0.371461, -1.418826, -2.541383, -0.752180, 1.570796, 1.942258],accel_mss,speed_ms,0,blend_radius_m)
      movel([0.370945, -1.419427, -2.540925, -0.752037, 1.570796, 1.941742],accel_mss,speed_ms,0,blend_radius_m)
      movel([0.370416, -1.420023, -2.540469, -0.751896, 1.570796, 1.941213],accel_mss,speed_ms,0,blend_radius_m)
      movel([0.369880, -1.420611, -2.540020, -0.751758, 1.570796, 1.940676],accel_mss,speed_ms,0,blend_radius_m)
      movel([0.369333, -1.421194, -2.539574, -0.751621, 1.570796, 1.940129],accel_mss,speed_ms,0,blend_radius_m)
      movel([0.368778, -1.421770, -2.539132, -0.751487, 1.570796, 1.939574],accel_mss,speed_ms,0,blend_radius_m)
      movel([0.368090, -1.422463, -2.538600, -0.751325, 1.570796, 1.938887],accel_mss,speed_ms,0,blend_radius_m)
      movel([0.367394, -1.423148, -2.538074, -0.751167, 1.570796, 1.938190],accel_mss,speed_ms,0,blend_radius_m)
      movel([0.366684, -1.423824, -2.537554, -0.751011, 1.570796, 1.937480],accel_mss,speed_ms,0,blend_radius_m)
      movel([0.365967, -1.424491, -2.537041, -0.750858, 1.570796, 1.936763],accel_mss,speed_ms,0,blend_radius_m)
      movel([0.365237, -1.425149, -2.536533, -0.750707, 1.570796, 1.936033],accel_mss,speed_ms,0,blend_radius_m)
      movel([0.364499, -1.425797, -2.536032, -0.750560, 1.570796, 1.935295],accel_mss,speed_ms,0,blend_radius_m)
      movel([0.363757, -1.426432, -2.535541, -0.750416, 1.570796, 1.934554],accel_mss,speed_ms,0,blend_radius_m)
      movel([0.363004, -1.427056, -2.535058, -0.750275, 1.570796, 1.933800],accel_mss,speed_ms,0,blend_radius_m)
      movel([0.362244, -1.427670, -2.534582, -0.750137, 1.570796, 1.933040],accel_mss,speed_ms,0,blend_radius_m)
      movel([0.361476, -1.428273, -2.534114, -0.750002, 1.570796, 1.932272],accel_mss,speed_ms,0,blend_radius_m)
      movel([0.360700, -1.428866, -2.533653, -0.749870, 1.570796, 1.931496],accel_mss,speed_ms,0,blend_radius_m)
      movel([0.359919, -1.429446, -2.533202, -0.749741, 1.570796, 1.930715],accel_mss,speed_ms,0,blend_radius_m)
      movel([0.359276, -1.429910, -2.532841, -0.749638, 1.570796, 1.930072],accel_mss,speed_ms,0,blend_radius_m)
      movel([0.358630, -1.430361, -2.532489, -0.749539, 1.570796, 1.929426],accel_mss,speed_ms,0,blend_radius_m)
      movel([0.357976, -1.430806, -2.532142, -0.749441, 1.570796, 1.928772],accel_mss,speed_ms,0,blend_radius_m)
      movel([0.357318, -1.431239, -2.531804, -0.749346, 1.570796, 1.928115],accel_mss,speed_ms,0,blend_radius_m)
      movel([0.356656, -1.431664, -2.531472, -0.749253, 1.570796, 1.927452],accel_mss,speed_ms,0,blend_radius_m)
      movel([0.355989, -1.432078, -2.531148, -0.749163, 1.570796, 1.926785],accel_mss,speed_ms,0,blend_radius_m)
      movel([0.355319, -1.432480, -2.530834, -0.749075, 1.570796, 1.926115],accel_mss,speed_ms,0,blend_radius_m)
      movel([0.354602, -1.432898, -2.530506, -0.748985, 1.570796, 1.925398],accel_mss,speed_ms,0,blend_radius_m)
      movel([0.353883, -1.433304, -2.530188, -0.748897, 1.570796, 1.924679],accel_mss,speed_ms,0,blend_radius_m)
      movel([0.353161, -1.433697, -2.529879, -0.748812, 1.570796, 1.923957],accel_mss,speed_ms,0,blend_radius_m)
      movel([0.352435, -1.434081, -2.529578, -0.748730, 1.570796, 1.923231],accel_mss,speed_ms,0,blend_radius_m)
      movel([0.351705, -1.434452, -2.529287, -0.748650, 1.570796, 1.922501],accel_mss,speed_ms,0,blend_radius_m)
      movel([0.350973, -1.434813, -2.529003, -0.748573, 1.570796, 1.921769],accel_mss,speed_ms,0,blend_radius_m)
      movel([0.350237, -1.435163, -2.528728, -0.748498, 1.570796, 1.921034],accel_mss,speed_ms,0,blend_radius_m)
      movel([0.349519, -1.435491, -2.528470, -0.748429, 1.570796, 1.920316],accel_mss,speed_ms,0,blend_radius_m)
      movel([0.348797, -1.435807, -2.528221, -0.748361, 1.570796, 1.919594],accel_mss,speed_ms,0,blend_radius_m)
      movel([0.348077, -1.436109, -2.527983, -0.748298, 1.570796, 1.918873],accel_mss,speed_ms,0,blend_radius_m)
      movel([0.347353, -1.436399, -2.527754, -0.748236, 1.570796, 1.918149],accel_mss,speed_ms,0,blend_radius_m)
      movel([0.346627, -1.436677, -2.527535, -0.748178, 1.570796, 1.917424],accel_mss,speed_ms,0,blend_radius_m)
      movel([0.345903, -1.436940, -2.527327, -0.748122, 1.570796, 1.916699],accel_mss,speed_ms,0,blend_radius_m)
      movel([0.345177, -1.437192, -2.527128, -0.748069, 1.570796, 1.915974],accel_mss,speed_ms,0,blend_radius_m)
      movel([0.344453, -1.437430, -2.526940, -0.748019, 1.570796, 1.915249],accel_mss,speed_ms,0,blend_radius_m)
      movel([0.343728, -1.437654, -2.526763, -0.747972, 1.570796, 1.914524],accel_mss,speed_ms,0,blend_radius_m)
      movel([0.343003, -1.437865, -2.526595, -0.747928, 1.570796, 1.913799],accel_mss,speed_ms,0,blend_radius_m)
      movel([0.342281, -1.438063, -2.526439, -0.747887, 1.570796, 1.913078],accel_mss,speed_ms,0,blend_radius_m)
      movel([0.341559, -1.438247, -2.526294, -0.747849, 1.570796, 1.912355],accel_mss,speed_ms,0,blend_radius_m)
      movel([0.340840, -1.438416, -2.526159, -0.747813, 1.570796, 1.911636],accel_mss,speed_ms,0,blend_radius_m)
      movel([0.340122, -1.438572, -2.526036, -0.747781, 1.570796, 1.910919],accel_mss,speed_ms,0,blend_radius_m)
      movel([0.339389, -1.438719, -2.525920, -0.747750, 1.570796, 1.910185],accel_mss,speed_ms,0,blend_radius_m)
      movel([0.338657, -1.438853, -2.525813, -0.747722, 1.570796, 1.909454],accel_mss,speed_ms,0,blend_radius_m)
      movel([0.337929, -1.438974, -2.525717, -0.747697, 1.570796, 1.908726],accel_mss,speed_ms,0,blend_radius_m)
      movel([0.337205, -1.439081, -2.525633, -0.747675, 1.570796, 1.908001],accel_mss,speed_ms,0,blend_radius_m)
      movel([0.336484, -1.439176, -2.525558, -0.747656, 1.570796, 1.907281],accel_mss,speed_ms,0,blend_radius_m)
      movel([0.335767, -1.439256, -2.525494, -0.747639, 1.570796, 1.906564],accel_mss,speed_ms,0,blend_radius_m)
      movel([0.335053, -1.439323, -2.525441, -0.747625, 1.570796, 1.905850],accel_mss,speed_ms,0,blend_radius_m)
      movel([0.334471, -1.439368, -2.525405, -0.747616, 1.570796, 1.905268],accel_mss,speed_ms,0,blend_radius_m)
      movel([0.333891, -1.439402, -2.525378, -0.747609, 1.570796, 1.904687],accel_mss,speed_ms,0,blend_radius_m)
      movel([0.333315, -1.439425, -2.525360, -0.747604, 1.570796, 1.904111],accel_mss,speed_ms,0,blend_radius_m)
      movel([0.332675, -1.439442, -2.525346, -0.747600, 1.570796, 1.903472],accel_mss,speed_ms,0,blend_radius_m)
      movel([0.332042, -1.439450, -2.525340, -0.747599, 1.570796, 1.902838],accel_mss,speed_ms,0,blend_radius_m)
      movel([0.331409, -1.439450, -2.525340, -0.747599, 1.570796, 1.902205],accel_mss,speed_ms,0,blend_radius_m)
      movel([0.330513, -1.439440, -2.525348, -0.747601, 1.570796, 1.901310],accel_mss,speed_ms,0,blend_radius_m)
      movel([0.329623, -1.439422, -2.525362, -0.747605, 1.570796, 1.900419],accel_mss,speed_ms,0,blend_radius_m)
      movel([0.329543, -1.439414, -2.525369, -0.747606, 1.570796, 1.900340],accel_mss,speed_ms,0,blend_radius_m)
      movel([0.329470, -1.439396, -2.525383, -0.747610, 1.570796, 1.900266],accel_mss,speed_ms,0,blend_radius_m)
      movel([0.329407, -1.439366, -2.525406, -0.747616, 1.570796, 1.900203],accel_mss,speed_ms,0,blend_radius_m)
      movel([0.329350, -1.439327, -2.525438, -0.747624, 1.570796, 1.900146],accel_mss,speed_ms,0,blend_radius_m)
      movel([0.329307, -1.439278, -2.525476, -0.747634, 1.570796, 1.900103],accel_mss,speed_ms,0,blend_radius_m)
      movel([0.329287, -1.439237, -2.525509, -0.747643, 1.570796, 1.900083],accel_mss,speed_ms,0,blend_radius_m)
      movel([0.329286, -1.439186, -2.525549, -0.747653, 1.570796, 1.900082],accel_mss,speed_ms,0,blend_radius_m)
      movel([0.329301, -1.439133, -2.525592, -0.747665, 1.570796, 1.900098],accel_mss,speed_ms,0,blend_radius_m)
      movel([0.335161, -1.426497, -2.535491, -0.750401, 1.570796, 1.905958],accel_mss,speed_ms,0,blend_radius_m)
      movel([0.340860, -1.414323, -2.544801, -0.753264, 1.570796, 1.911656],accel_mss,speed_ms,0,blend_radius_m)
      movel([0.341139, -1.413743, -2.545239, -0.753406, 1.570796, 1.911936],accel_mss,speed_ms,0,blend_radius_m)
      movel([0.341435, -1.413162, -2.545678, -0.753549, 1.570796, 1.912232],accel_mss,speed_ms,0,blend_radius_m)
      movel([0.341746, -1.412581, -2.546116, -0.753692, 1.570796, 1.912543],accel_mss,speed_ms,0,blend_radius_m)
      movel([0.342131, -1.411877, -2.546645, -0.753866, 1.570796, 1.912927],accel_mss,speed_ms,0,blend_radius_m)
      movel([0.358719, -1.412778, -2.545967, -0.753644, 1.570796, 1.929516],accel_mss,speed_ms,0,blend_radius_m)
      movel([0.365044, -1.413195, -2.545653, -0.753541, 1.570796, 1.935840],accel_mss,speed_ms,0,blend_radius_m)
      movel([0.370351, -1.413582, -2.545361, -0.753446, 1.570796, 1.941147],accel_mss,speed_ms,0,blend_radius_m)
      movel([0.375158, -1.413958, -2.545077, -0.753354, 1.570796, 1.945954],accel_mss,speed_ms,0,blend_radius_m)
      speed_ms = 0.003
      movel([0.375158, -1.417147, -2.546510, -0.748732, 1.570796, 1.945954],accel_mss,speed_ms,0,blend_radius_m)
      speed_ms = 0.007
      movel([0.375180, -1.417153, -2.546506, -0.748730, 1.570796, 1.945976],accel_mss,speed_ms,0,blend_radius_m)
      movel([0.375195, -1.417163, -2.546498, -0.748728, 1.570796, 1.945992],accel_mss,speed_ms,0,blend_radius_m)
      movel([0.375198, -1.417185, -2.546482, -0.748723, 1.570796, 1.945994],accel_mss,speed_ms,0,blend_radius_m)
      movel([0.375187, -1.417206, -2.546465, -0.748717, 1.570796, 1.945983],accel_mss,speed_ms,0,blend_radius_m)
      movel([0.374177, -1.418562, -2.545435, -0.748392, 1.570796, 1.944973],accel_mss,speed_ms,0,blend_radius_m)
      movel([0.373704, -1.419192, -2.544955, -0.748242, 1.570796, 1.944500],accel_mss,speed_ms,0,blend_radius_m)
      movel([0.373225, -1.419820, -2.544476, -0.748093, 1.570796, 1.944021],accel_mss,speed_ms,0,blend_radius_m)
      movel([0.372848, -1.420308, -2.544104, -0.747977, 1.570796, 1.943644],accel_mss,speed_ms,0,blend_radius_m)
      movel([0.372466, -1.420789, -2.543737, -0.747864, 1.570796, 1.943262],accel_mss,speed_ms,0,blend_radius_m)
      movel([0.371969, -1.421399, -2.543270, -0.747720, 1.570796, 1.942765],accel_mss,speed_ms,0,blend_radius_m)
      movel([0.371461, -1.422002, -2.542808, -0.747579, 1.570796, 1.942258],accel_mss,speed_ms,0,blend_radius_m)
      movel([0.370945, -1.422601, -2.542349, -0.747439, 1.570796, 1.941742],accel_mss,speed_ms,0,blend_radius_m)
      movel([0.370416, -1.423196, -2.541892, -0.747301, 1.570796, 1.941213],accel_mss,speed_ms,0,blend_radius_m)
      movel([0.369880, -1.423781, -2.541442, -0.747165, 1.570796, 1.940676],accel_mss,speed_ms,0,blend_radius_m)
      movel([0.369333, -1.424363, -2.540995, -0.747031, 1.570796, 1.940129],accel_mss,speed_ms,0,blend_radius_m)
      movel([0.368778, -1.424938, -2.540552, -0.746899, 1.570796, 1.939574],accel_mss,speed_ms,0,blend_radius_m)
      movel([0.368090, -1.425629, -2.540019, -0.746741, 1.570796, 1.938887],accel_mss,speed_ms,0,blend_radius_m)
      movel([0.367394, -1.426311, -2.539492, -0.746585, 1.570796, 1.938190],accel_mss,speed_ms,0,blend_radius_m)
      movel([0.366684, -1.426985, -2.538971, -0.746433, 1.570796, 1.937480],accel_mss,speed_ms,0,blend_radius_m)
      movel([0.365967, -1.427650, -2.538457, -0.746282, 1.570796, 1.936763],accel_mss,speed_ms,0,blend_radius_m)
      movel([0.365237, -1.428307, -2.537948, -0.746135, 1.570796, 1.936033],accel_mss,speed_ms,0,blend_radius_m)
      movel([0.364499, -1.428952, -2.537446, -0.745990, 1.570796, 1.935295],accel_mss,speed_ms,0,blend_radius_m)
      movel([0.363757, -1.429586, -2.536954, -0.745849, 1.570796, 1.934554],accel_mss,speed_ms,0,blend_radius_m)
      movel([0.363004, -1.430208, -2.536470, -0.745711, 1.570796, 1.933800],accel_mss,speed_ms,0,blend_radius_m)
      movel([0.362244, -1.430820, -2.535993, -0.745576, 1.570796, 1.933040],accel_mss,speed_ms,0,blend_radius_m)
      movel([0.361476, -1.431422, -2.535524, -0.745443, 1.570796, 1.932272],accel_mss,speed_ms,0,blend_radius_m)
      movel([0.360700, -1.432013, -2.535062, -0.745314, 1.570796, 1.931496],accel_mss,speed_ms,0,blend_radius_m)
      movel([0.359919, -1.432591, -2.534610, -0.745188, 1.570796, 1.930715],accel_mss,speed_ms,0,blend_radius_m)
      movel([0.359276, -1.433054, -2.534248, -0.745087, 1.570796, 1.930072],accel_mss,speed_ms,0,blend_radius_m)
      movel([0.358630, -1.433504, -2.533896, -0.744989, 1.570796, 1.929426],accel_mss,speed_ms,0,blend_radius_m)
      movel([0.357976, -1.433948, -2.533548, -0.744894, 1.570796, 1.928772],accel_mss,speed_ms,0,blend_radius_m)
      movel([0.357318, -1.434379, -2.533209, -0.744801, 1.570796, 1.928115],accel_mss,speed_ms,0,blend_radius_m)
      movel([0.356656, -1.434803, -2.532877, -0.744710, 1.570796, 1.927452],accel_mss,speed_ms,0,blend_radius_m)
      movel([0.355989, -1.435216, -2.532552, -0.744621, 1.570796, 1.926785],accel_mss,speed_ms,0,blend_radius_m)
      movel([0.355319, -1.435617, -2.532237, -0.744536, 1.570796, 1.926115],accel_mss,speed_ms,0,blend_radius_m)
      movel([0.354602, -1.436033, -2.531909, -0.744447, 1.570796, 1.925398],accel_mss,speed_ms,0,blend_radius_m)
      movel([0.353883, -1.436438, -2.531590, -0.744361, 1.570796, 1.924679],accel_mss,speed_ms,0,blend_radius_m)
      movel([0.353161, -1.436830, -2.531281, -0.744278, 1.570796, 1.923957],accel_mss,speed_ms,0,blend_radius_m)
      movel([0.352435, -1.437213, -2.530979, -0.744197, 1.570796, 1.923231],accel_mss,speed_ms,0,blend_radius_m)
      movel([0.351705, -1.437583, -2.530687, -0.744119, 1.570796, 1.922501],accel_mss,speed_ms,0,blend_radius_m)
      movel([0.350973, -1.437943, -2.530402, -0.744043, 1.570796, 1.921769],accel_mss,speed_ms,0,blend_radius_m)
      movel([0.350237, -1.438291, -2.530127, -0.743971, 1.570796, 1.921034],accel_mss,speed_ms,0,blend_radius_m)
      movel([0.349519, -1.438618, -2.529868, -0.743902, 1.570796, 1.920316],accel_mss,speed_ms,0,blend_radius_m)
      movel([0.348797, -1.438934, -2.529619, -0.743837, 1.570796, 1.919594],accel_mss,speed_ms,0,blend_radius_m)
      movel([0.348077, -1.439235, -2.529380, -0.743774, 1.570796, 1.918873],accel_mss,speed_ms,0,blend_radius_m)
      movel([0.347353, -1.439524, -2.529151, -0.743714, 1.570796, 1.918149],accel_mss,speed_ms,0,blend_radius_m)
      movel([0.346627, -1.439801, -2.528932, -0.743657, 1.570796, 1.917424],accel_mss,speed_ms,0,blend_radius_m)
      movel([0.345903, -1.440064, -2.528723, -0.743602, 1.570796, 1.916699],accel_mss,speed_ms,0,blend_radius_m)
      movel([0.345177, -1.440315, -2.528524, -0.743550, 1.570796, 1.915974],accel_mss,speed_ms,0,blend_radius_m)
      movel([0.344453, -1.440552, -2.528335, -0.743502, 1.570796, 1.915249],accel_mss,speed_ms,0,blend_radius_m)
      movel([0.343728, -1.440775, -2.528158, -0.743456, 1.570796, 1.914524],accel_mss,speed_ms,0,blend_radius_m)
      movel([0.343003, -1.440986, -2.527990, -0.743412, 1.570796, 1.913799],accel_mss,speed_ms,0,blend_radius_m)
      movel([0.342281, -1.441183, -2.527834, -0.743372, 1.570796, 1.913078],accel_mss,speed_ms,0,blend_radius_m)
      movel([0.341559, -1.441367, -2.527688, -0.743334, 1.570796, 1.912355],accel_mss,speed_ms,0,blend_radius_m)
      movel([0.340840, -1.441536, -2.527553, -0.743300, 1.570796, 1.911636],accel_mss,speed_ms,0,blend_radius_m)
      movel([0.340122, -1.441691, -2.527430, -0.743268, 1.570796, 1.910919],accel_mss,speed_ms,0,blend_radius_m)
      movel([0.339389, -1.441837, -2.527313, -0.743238, 1.570796, 1.910185],accel_mss,speed_ms,0,blend_radius_m)
      movel([0.338657, -1.441971, -2.527206, -0.743211, 1.570796, 1.909454],accel_mss,speed_ms,0,blend_radius_m)
      movel([0.337929, -1.442092, -2.527111, -0.743187, 1.570796, 1.908726],accel_mss,speed_ms,0,blend_radius_m)
      movel([0.337205, -1.442198, -2.527026, -0.743165, 1.570796, 1.908001],accel_mss,speed_ms,0,blend_radius_m)
      movel([0.336484, -1.442293, -2.526951, -0.743146, 1.570796, 1.907281],accel_mss,speed_ms,0,blend_radius_m)
      movel([0.335767, -1.442373, -2.526886, -0.743129, 1.570796, 1.906564],accel_mss,speed_ms,0,blend_radius_m)
      movel([0.335053, -1.442440, -2.526833, -0.743116, 1.570796, 1.905850],accel_mss,speed_ms,0,blend_radius_m)
      movel([0.334471, -1.442484, -2.526798, -0.743107, 1.570796, 1.905268],accel_mss,speed_ms,0,blend_radius_m)
      movel([0.333891, -1.442519, -2.526771, -0.743100, 1.570796, 1.904687],accel_mss,speed_ms,0,blend_radius_m)
      movel([0.333315, -1.442541, -2.526753, -0.743095, 1.570796, 1.904111],accel_mss,speed_ms,0,blend_radius_m)
      movel([0.332675, -1.442559, -2.526739, -0.743092, 1.570796, 1.903472],accel_mss,speed_ms,0,blend_radius_m)
      movel([0.332042, -1.442566, -2.526732, -0.743090, 1.570796, 1.902838],accel_mss,speed_ms,0,blend_radius_m)
      movel([0.331409, -1.442566, -2.526732, -0.743090, 1.570796, 1.902205],accel_mss,speed_ms,0,blend_radius_m)
      movel([0.330513, -1.442556, -2.526741, -0.743092, 1.570796, 1.901310],accel_mss,speed_ms,0,blend_radius_m)
      movel([0.329623, -1.442538, -2.526755, -0.743096, 1.570796, 1.900419],accel_mss,speed_ms,0,blend_radius_m)
      movel([0.329543, -1.442530, -2.526761, -0.743098, 1.570796, 1.900340],accel_mss,speed_ms,0,blend_radius_m)
      movel([0.329470, -1.442512, -2.526776, -0.743101, 1.570796, 1.900266],accel_mss,speed_ms,0,blend_radius_m)
      movel([0.329407, -1.442483, -2.526799, -0.743107, 1.570796, 1.900203],accel_mss,speed_ms,0,blend_radius_m)
      movel([0.329350, -1.442443, -2.526830, -0.743115, 1.570796, 1.900146],accel_mss,speed_ms,0,blend_radius_m)
      movel([0.329307, -1.442395, -2.526869, -0.743125, 1.570796, 1.900103],accel_mss,speed_ms,0,blend_radius_m)
      movel([0.329287, -1.442354, -2.526902, -0.743133, 1.570796, 1.900083],accel_mss,speed_ms,0,blend_radius_m)
      movel([0.329286, -1.442303, -2.526942, -0.743144, 1.570796, 1.900082],accel_mss,speed_ms,0,blend_radius_m)
      movel([0.329301, -1.442250, -2.526985, -0.743154, 1.570796, 1.900098],accel_mss,speed_ms,0,blend_radius_m)
      movel([0.335161, -1.429651, -2.536903, -0.745835, 1.570796, 1.905958],accel_mss,speed_ms,0,blend_radius_m)
      movel([0.340860, -1.417512, -2.546233, -0.748644, 1.570796, 1.911656],accel_mss,speed_ms,0,blend_radius_m)
      movel([0.341139, -1.416933, -2.546672, -0.748783, 1.570796, 1.911936],accel_mss,speed_ms,0,blend_radius_m)
      movel([0.341435, -1.416354, -2.547112, -0.748923, 1.570796, 1.912232],accel_mss,speed_ms,0,blend_radius_m)
      movel([0.341746, -1.415774, -2.547551, -0.749064, 1.570796, 1.912543],accel_mss,speed_ms,0,blend_radius_m)
      movel([0.342131, -1.415073, -2.548081, -0.749235, 1.570796, 1.912927],accel_mss,speed_ms,0,blend_radius_m)
      movel([0.358719, -1.415971, -2.547402, -0.749016, 1.570796, 1.929516],accel_mss,speed_ms,0,blend_radius_m)
      movel([0.365044, -1.416387, -2.547087, -0.748915, 1.570796, 1.935840],accel_mss,speed_ms,0,blend_radius_m)
      movel([0.370351, -1.416773, -2.546794, -0.748822, 1.570796, 1.941147],accel_mss,speed_ms,0,blend_radius_m)
      movel([0.375158, -1.417147, -2.546510, -0.748732, 1.570796, 1.945954],accel_mss,speed_ms,0,blend_radius_m)
      speed_ms = 0.003
      movel([0.375158, -1.404512, -2.540729, -0.767148, 1.570796, 1.945954],accel_mss,speed_ms,0,blend_radius_m)
      speed_ms = 0.01
      movel([0.375158, -1.380220, -2.528774, -0.803396, 1.570796, 1.945954],accel_mss,speed_ms,0,blend_radius_m)
      movel([0.335045, -1.431374, -2.490212, -0.790803, 1.570796, 1.905842],accel_mss,speed_ms,0,blend_radius_m)
      movel([0.335045, -1.454665, -2.501542, -0.756183, 1.570796, 1.905842],accel_mss,speed_ms,0,blend_radius_m)
      speed_ms = 0.003
      movel([0.335045, -1.463693, -2.505656, -0.743040, 1.570796, 1.905842],accel_mss,speed_ms,0,blend_radius_m)
      speed_ms = 0.007
      movel([0.335236, -1.463780, -2.505584, -0.743026, 1.570796, 1.906033],accel_mss,speed_ms,0,blend_radius_m)
      movel([0.335250, -1.463793, -2.505573, -0.743023, 1.570796, 1.906047],accel_mss,speed_ms,0,blend_radius_m)
      movel([0.335257, -1.463810, -2.505558, -0.743020, 1.570796, 1.906053],accel_mss,speed_ms,0,blend_radius_m)
      movel([0.335252, -1.463834, -2.505538, -0.743016, 1.570796, 1.906048],accel_mss,speed_ms,0,blend_radius_m)
      movel([0.335233, -1.463878, -2.505502, -0.743009, 1.570796, 1.906030],accel_mss,speed_ms,0,blend_radius_m)
      movel([0.335208, -1.463925, -2.505463, -0.743001, 1.570796, 1.906004],accel_mss,speed_ms,0,blend_radius_m)
      movel([0.334086, -1.465654, -2.504024, -0.742711, 1.570796, 1.904882],accel_mss,speed_ms,0,blend_radius_m)
      movel([0.332832, -1.467586, -2.502410, -0.742392, 1.570796, 1.903629],accel_mss,speed_ms,0,blend_radius_m)
      movel([0.331361, -1.469852, -2.500511, -0.742026, 1.570796, 1.902157],accel_mss,speed_ms,0,blend_radius_m)
      movel([0.329888, -1.472109, -2.498611, -0.741669, 1.570796, 1.900684],accel_mss,speed_ms,0,blend_radius_m)
      movel([0.328639, -1.474014, -2.497001, -0.741374, 1.570796, 1.899435],accel_mss,speed_ms,0,blend_radius_m)
      movel([0.327523, -1.475713, -2.495561, -0.741116, 1.570796, 1.898320],accel_mss,speed_ms,0,blend_radius_m)
      movel([0.327493, -1.475751, -2.495528, -0.741110, 1.570796, 1.898289],accel_mss,speed_ms,0,blend_radius_m)
      movel([0.327456, -1.475783, -2.495501, -0.741105, 1.570796, 1.898252],accel_mss,speed_ms,0,blend_radius_m)
      movel([0.327430, -1.475798, -2.495488, -0.741103, 1.570796, 1.898226],accel_mss,speed_ms,0,blend_radius_m)
      movel([0.327404, -1.475804, -2.495483, -0.741102, 1.570796, 1.898201],accel_mss,speed_ms,0,blend_radius_m)
      movel([0.327379, -1.475806, -2.495482, -0.741102, 1.570796, 1.898175],accel_mss,speed_ms,0,blend_radius_m)
      movel([0.326884, -1.475727, -2.495548, -0.741114, 1.570796, 1.897681],accel_mss,speed_ms,0,blend_radius_m)
      movel([0.326600, -1.475677, -2.495591, -0.741121, 1.570796, 1.897397],accel_mss,speed_ms,0,blend_radius_m)
      movel([0.326315, -1.475625, -2.495635, -0.741129, 1.570796, 1.897111],accel_mss,speed_ms,0,blend_radius_m)
      movel([0.325658, -1.475488, -2.495751, -0.741150, 1.570796, 1.896454],accel_mss,speed_ms,0,blend_radius_m)
      movel([0.315472, -1.473531, -2.497410, -0.741448, 1.570796, 1.886268],accel_mss,speed_ms,0,blend_radius_m)
      movel([0.313321, -1.473128, -2.497750, -0.741511, 1.570796, 1.884118],accel_mss,speed_ms,0,blend_radius_m)
      movel([0.311172, -1.472720, -2.498095, -0.741574, 1.570796, 1.881969],accel_mss,speed_ms,0,blend_radius_m)
      movel([0.310041, -1.472501, -2.498280, -0.741608, 1.570796, 1.880837],accel_mss,speed_ms,0,blend_radius_m)
      movel([0.308911, -1.472274, -2.498472, -0.741643, 1.570796, 1.879708],accel_mss,speed_ms,0,blend_radius_m)
      movel([0.307788, -1.472037, -2.498671, -0.741680, 1.570796, 1.878585],accel_mss,speed_ms,0,blend_radius_m)
      movel([0.306670, -1.471792, -2.498878, -0.741719, 1.570796, 1.877466],accel_mss,speed_ms,0,blend_radius_m)
      movel([0.305780, -1.471588, -2.499050, -0.741751, 1.570796, 1.876576],accel_mss,speed_ms,0,blend_radius_m)
      movel([0.304894, -1.471375, -2.499229, -0.741784, 1.570796, 1.875691],accel_mss,speed_ms,0,blend_radius_m)
      movel([0.304016, -1.471153, -2.499417, -0.741819, 1.570796, 1.874812],accel_mss,speed_ms,0,blend_radius_m)
      movel([0.303144, -1.470921, -2.499612, -0.741856, 1.570796, 1.873940],accel_mss,speed_ms,0,blend_radius_m)
      movel([0.302323, -1.470693, -2.499804, -0.741892, 1.570796, 1.873120],accel_mss,speed_ms,0,blend_radius_m)
      movel([0.301510, -1.470453, -2.500006, -0.741930, 1.570796, 1.872307],accel_mss,speed_ms,0,blend_radius_m)
      movel([0.300704, -1.470203, -2.500216, -0.741970, 1.570796, 1.871500],accel_mss,speed_ms,0,blend_radius_m)
      movel([0.299905, -1.469942, -2.500435, -0.742012, 1.570796, 1.870702],accel_mss,speed_ms,0,blend_radius_m)
      movel([0.299196, -1.469695, -2.500642, -0.742051, 1.570796, 1.869992],accel_mss,speed_ms,0,blend_radius_m)
      movel([0.298496, -1.469437, -2.500860, -0.742093, 1.570796, 1.869293],accel_mss,speed_ms,0,blend_radius_m)
      movel([0.297805, -1.469166, -2.501087, -0.742136, 1.570796, 1.868601],accel_mss,speed_ms,0,blend_radius_m)
      movel([0.297126, -1.468880, -2.501327, -0.742182, 1.570796, 1.867922],accel_mss,speed_ms,0,blend_radius_m)
      movel([0.296454, -1.468584, -2.501575, -0.742230, 1.570796, 1.867251],accel_mss,speed_ms,0,blend_radius_m)
      movel([0.295795, -1.468274, -2.501835, -0.742280, 1.570796, 1.866592],accel_mss,speed_ms,0,blend_radius_m)
      movel([0.295324, -1.468037, -2.502033, -0.742319, 1.570796, 1.866120],accel_mss,speed_ms,0,blend_radius_m)
      movel([0.294866, -1.467787, -2.502243, -0.742360, 1.570796, 1.865662],accel_mss,speed_ms,0,blend_radius_m)
      movel([0.294417, -1.467526, -2.502461, -0.742402, 1.570796, 1.865213],accel_mss,speed_ms,0,blend_radius_m)
      movel([0.293983, -1.467250, -2.502691, -0.742447, 1.570796, 1.864779],accel_mss,speed_ms,0,blend_radius_m)
      movel([0.293559, -1.466963, -2.502932, -0.742495, 1.570796, 1.864355],accel_mss,speed_ms,0,blend_radius_m)
      movel([0.293149, -1.466663, -2.503182, -0.742544, 1.570796, 1.863946],accel_mss,speed_ms,0,blend_radius_m)
      movel([0.292750, -1.466350, -2.503443, -0.742595, 1.570796, 1.863546],accel_mss,speed_ms,0,blend_radius_m)
      movel([0.292420, -1.466070, -2.503677, -0.742642, 1.570796, 1.863216],accel_mss,speed_ms,0,blend_radius_m)
      movel([0.292102, -1.465776, -2.503922, -0.742691, 1.570796, 1.862898],accel_mss,speed_ms,0,blend_radius_m)
      movel([0.291798, -1.465472, -2.504175, -0.742741, 1.570796, 1.862595],accel_mss,speed_ms,0,blend_radius_m)
      movel([0.291509, -1.465156, -2.504439, -0.742794, 1.570796, 1.862305],accel_mss,speed_ms,0,blend_radius_m)
      movel([0.291236, -1.464828, -2.504712, -0.742849, 1.570796, 1.862032],accel_mss,speed_ms,0,blend_radius_m)
      movel([0.290975, -1.464488, -2.504995, -0.742906, 1.570796, 1.861771],accel_mss,speed_ms,0,blend_radius_m)
      movel([0.290729, -1.464138, -2.505286, -0.742965, 1.570796, 1.861525],accel_mss,speed_ms,0,blend_radius_m)
      movel([0.290549, -1.463852, -2.505524, -0.743013, 1.570796, 1.861346],accel_mss,speed_ms,0,blend_radius_m)
      movel([0.290383, -1.463556, -2.505769, -0.743063, 1.570796, 1.861180],accel_mss,speed_ms,0,blend_radius_m)
      movel([0.290233, -1.463252, -2.506022, -0.743115, 1.570796, 1.861029],accel_mss,speed_ms,0,blend_radius_m)
      movel([0.290095, -1.462938, -2.506282, -0.743169, 1.570796, 1.860892],accel_mss,speed_ms,0,blend_radius_m)
      movel([0.289976, -1.462616, -2.506550, -0.743224, 1.570796, 1.860772],accel_mss,speed_ms,0,blend_radius_m)
      movel([0.289869, -1.462286, -2.506823, -0.743280, 1.570796, 1.860665],accel_mss,speed_ms,0,blend_radius_m)
      movel([0.289780, -1.461947, -2.507104, -0.743338, 1.570796, 1.860576],accel_mss,speed_ms,0,blend_radius_m)
      movel([0.289703, -1.461601, -2.507390, -0.743398, 1.570796, 1.860500],accel_mss,speed_ms,0,blend_radius_m)
      movel([0.289650, -1.461294, -2.507644, -0.743451, 1.570796, 1.860447],accel_mss,speed_ms,0,blend_radius_m)
      movel([0.289607, -1.460982, -2.507902, -0.743505, 1.570796, 1.860404],accel_mss,speed_ms,0,blend_radius_m)
      movel([0.289577, -1.460665, -2.508164, -0.743560, 1.570796, 1.860373],accel_mss,speed_ms,0,blend_radius_m)
      movel([0.289553, -1.460346, -2.508427, -0.743616, 1.570796, 1.860349],accel_mss,speed_ms,0,blend_radius_m)
      movel([0.289545, -1.460062, -2.508662, -0.743666, 1.570796, 1.860342],accel_mss,speed_ms,0,blend_radius_m)
      movel([0.289550, -1.459773, -2.508900, -0.743716, 1.570796, 1.860346],accel_mss,speed_ms,0,blend_radius_m)
      movel([0.289571, -1.459478, -2.509143, -0.743768, 1.570796, 1.860367],accel_mss,speed_ms,0,blend_radius_m)
      movel([0.289603, -1.459183, -2.509386, -0.743820, 1.570796, 1.860399],accel_mss,speed_ms,0,blend_radius_m)
      movel([0.289651, -1.458859, -2.509653, -0.743877, 1.570796, 1.860447],accel_mss,speed_ms,0,blend_radius_m)
      movel([0.289714, -1.458534, -2.509921, -0.743935, 1.570796, 1.860510],accel_mss,speed_ms,0,blend_radius_m)
      movel([0.289789, -1.458205, -2.510191, -0.743993, 1.570796, 1.860585],accel_mss,speed_ms,0,blend_radius_m)
      movel([0.289875, -1.457876, -2.510462, -0.744052, 1.570796, 1.860671],accel_mss,speed_ms,0,blend_radius_m)
      movel([0.290046, -1.457302, -2.510932, -0.744154, 1.570796, 1.860843],accel_mss,speed_ms,0,blend_radius_m)
      movel([0.290229, -1.456727, -2.511404, -0.744258, 1.570796, 1.861025],accel_mss,speed_ms,0,blend_radius_m)
      movel([0.290425, -1.456151, -2.511876, -0.744362, 1.570796, 1.861221],accel_mss,speed_ms,0,blend_radius_m)
      movel([0.290736, -1.455296, -2.512576, -0.744517, 1.570796, 1.861532],accel_mss,speed_ms,0,blend_radius_m)
      movel([0.290875, -1.454927, -2.512877, -0.744585, 1.570796, 1.861671],accel_mss,speed_ms,0,blend_radius_m)
      movel([0.291019, -1.454558, -2.513179, -0.744652, 1.570796, 1.861815],accel_mss,speed_ms,0,blend_radius_m)
      movel([0.291273, -1.453924, -2.513696, -0.744769, 1.570796, 1.862069],accel_mss,speed_ms,0,blend_radius_m)
      movel([0.291289, -1.453893, -2.513721, -0.744775, 1.570796, 1.862085],accel_mss,speed_ms,0,blend_radius_m)
      movel([0.291312, -1.453862, -2.513747, -0.744780, 1.570796, 1.862109],accel_mss,speed_ms,0,blend_radius_m)
      movel([0.291342, -1.453836, -2.513768, -0.744785, 1.570796, 1.862138],accel_mss,speed_ms,0,blend_radius_m)
      movel([0.291377, -1.453815, -2.513785, -0.744789, 1.570796, 1.862173],accel_mss,speed_ms,0,blend_radius_m)
      movel([0.291414, -1.453804, -2.513794, -0.744791, 1.570796, 1.862211],accel_mss,speed_ms,0,blend_radius_m)
      movel([0.291449, -1.453803, -2.513795, -0.744791, 1.570796, 1.862245],accel_mss,speed_ms,0,blend_radius_m)
      movel([0.297738, -1.455050, -2.512777, -0.744562, 1.570796, 1.868535],accel_mss,speed_ms,0,blend_radius_m)
      movel([0.301205, -1.455760, -2.512197, -0.744433, 1.570796, 1.872001],accel_mss,speed_ms,0,blend_radius_m)
      movel([0.304655, -1.456490, -2.511599, -0.744301, 1.570796, 1.875452],accel_mss,speed_ms,0,blend_radius_m)
      movel([0.308729, -1.457376, -2.510872, -0.744141, 1.570796, 1.879525],accel_mss,speed_ms,0,blend_radius_m)
      movel([0.312786, -1.458284, -2.510126, -0.743979, 1.570796, 1.883582],accel_mss,speed_ms,0,blend_radius_m)
      movel([0.320904, -1.460169, -2.508573, -0.743647, 1.570796, 1.891700],accel_mss,speed_ms,0,blend_radius_m)
      movel([0.327823, -1.461842, -2.507190, -0.743356, 1.570796, 1.898620],accel_mss,speed_ms,0,blend_radius_m)
      movel([0.333854, -1.463353, -2.505938, -0.743098, 1.570796, 1.904650],accel_mss,speed_ms,0,blend_radius_m)
      movel([0.334793, -1.463600, -2.505733, -0.743056, 1.570796, 1.905589],accel_mss,speed_ms,0,blend_radius_m)
      movel([0.334922, -1.463644, -2.505696, -0.743049, 1.570796, 1.905718],accel_mss,speed_ms,0,blend_radius_m)
      movel([0.335045, -1.463693, -2.505656, -0.743040, 1.570796, 1.905842],accel_mss,speed_ms,0,blend_radius_m)
      speed_ms = 0.003
      movel([0.335045, -1.466737, -2.507011, -0.738640, 1.570796, 1.905842],accel_mss,speed_ms,0,blend_radius_m)
      speed_ms = 0.007
      movel([0.335236, -1.466824, -2.506939, -0.738626, 1.570796, 1.906033],accel_mss,speed_ms,0,blend_radius_m)
      movel([0.335250, -1.466838, -2.506927, -0.738624, 1.570796, 1.906047],accel_mss,speed_ms,0,blend_radius_m)
      movel([0.335257, -1.466855, -2.506913, -0.738621, 1.570796, 1.906053],accel_mss,speed_ms,0,blend_radius_m)
      movel([0.335252, -1.466879, -2.506893, -0.738617, 1.570796, 1.906048],accel_mss,speed_ms,0,blend_radius_m)
      movel([0.335233, -1.466923, -2.506856, -0.738610, 1.570796, 1.906030],accel_mss,speed_ms,0,blend_radius_m)
      movel([0.335208, -1.466969, -2.506818, -0.738602, 1.570796, 1.906004],accel_mss,speed_ms,0,blend_radius_m)
      movel([0.334086, -1.468693, -2.505376, -0.738320, 1.570796, 1.904882],accel_mss,speed_ms,0,blend_radius_m)
      movel([0.332832, -1.470620, -2.503759, -0.738010, 1.570796, 1.903629],accel_mss,speed_ms,0,blend_radius_m)
      movel([0.331361, -1.472879, -2.501856, -0.737654, 1.570796, 1.902157],accel_mss,speed_ms,0,blend_radius_m)
      movel([0.329888, -1.475129, -2.499953, -0.737307, 1.570796, 1.900684],accel_mss,speed_ms,0,blend_radius_m)
      movel([0.328639, -1.477029, -2.498340, -0.737021, 1.570796, 1.899435],accel_mss,speed_ms,0,blend_radius_m)
      movel([0.327523, -1.478722, -2.496897, -0.736770, 1.570796, 1.898320],accel_mss,speed_ms,0,blend_radius_m)
      movel([0.327493, -1.478760, -2.496865, -0.736764, 1.570796, 1.898289],accel_mss,speed_ms,0,blend_radius_m)
      movel([0.327456, -1.478792, -2.496837, -0.736760, 1.570796, 1.898252],accel_mss,speed_ms,0,blend_radius_m)
      movel([0.327430, -1.478806, -2.496825, -0.736757, 1.570796, 1.898226],accel_mss,speed_ms,0,blend_radius_m)
      movel([0.327404, -1.478813, -2.496819, -0.736756, 1.570796, 1.898201],accel_mss,speed_ms,0,blend_radius_m)
      movel([0.327379, -1.478814, -2.496818, -0.736756, 1.570796, 1.898175],accel_mss,speed_ms,0,blend_radius_m)
      movel([0.326884, -1.478736, -2.496885, -0.736768, 1.570796, 1.897681],accel_mss,speed_ms,0,blend_radius_m)
      movel([0.326600, -1.478686, -2.496928, -0.736775, 1.570796, 1.897397],accel_mss,speed_ms,0,blend_radius_m)
      movel([0.326315, -1.478634, -2.496972, -0.736783, 1.570796, 1.897111],accel_mss,speed_ms,0,blend_radius_m)
      movel([0.325658, -1.478498, -2.497088, -0.736803, 1.570796, 1.896454],accel_mss,speed_ms,0,blend_radius_m)
      movel([0.315472, -1.476546, -2.498750, -0.737093, 1.570796, 1.886268],accel_mss,speed_ms,0,blend_radius_m)
      movel([0.313321, -1.476145, -2.499091, -0.737153, 1.570796, 1.884118],accel_mss,speed_ms,0,blend_radius_m)
      movel([0.311172, -1.475738, -2.499436, -0.737215, 1.570796, 1.881969],accel_mss,speed_ms,0,blend_radius_m)
      movel([0.310041, -1.475520, -2.499621, -0.737248, 1.570796, 1.880837],accel_mss,speed_ms,0,blend_radius_m)
      movel([0.308911, -1.475293, -2.499814, -0.737282, 1.570796, 1.879708],accel_mss,speed_ms,0,blend_radius_m)
      movel([0.307788, -1.475057, -2.500014, -0.737318, 1.570796, 1.878585],accel_mss,speed_ms,0,blend_radius_m)
      movel([0.306670, -1.474813, -2.500221, -0.737355, 1.570796, 1.877466],accel_mss,speed_ms,0,blend_radius_m)
      movel([0.305780, -1.474610, -2.500393, -0.737386, 1.570796, 1.876576],accel_mss,speed_ms,0,blend_radius_m)
      movel([0.304894, -1.474397, -2.500573, -0.737419, 1.570796, 1.875691],accel_mss,speed_ms,0,blend_radius_m)
      movel([0.304016, -1.474176, -2.500760, -0.737453, 1.570796, 1.874812],accel_mss,speed_ms,0,blend_radius_m)
      movel([0.303144, -1.473944, -2.500956, -0.737489, 1.570796, 1.873940],accel_mss,speed_ms,0,blend_radius_m)
      movel([0.302323, -1.473717, -2.501148, -0.737524, 1.570796, 1.873120],accel_mss,speed_ms,0,blend_radius_m)
      movel([0.301510, -1.473477, -2.501351, -0.737561, 1.570796, 1.872307],accel_mss,speed_ms,0,blend_radius_m)
      movel([0.300704, -1.473229, -2.501561, -0.737599, 1.570796, 1.871500],accel_mss,speed_ms,0,blend_radius_m)
      movel([0.299905, -1.472969, -2.501780, -0.737640, 1.570796, 1.870702],accel_mss,speed_ms,0,blend_radius_m)
      movel([0.299196, -1.472723, -2.501988, -0.737678, 1.570796, 1.869992],accel_mss,speed_ms,0,blend_radius_m)
      movel([0.298496, -1.472465, -2.502206, -0.737719, 1.570796, 1.869293],accel_mss,speed_ms,0,blend_radius_m)
      movel([0.297805, -1.472195, -2.502433, -0.737761, 1.570796, 1.868601],accel_mss,speed_ms,0,blend_radius_m)
      movel([0.297126, -1.471909, -2.502674, -0.737806, 1.570796, 1.867922],accel_mss,speed_ms,0,blend_radius_m)
      movel([0.296454, -1.471614, -2.502923, -0.737852, 1.570796, 1.867251],accel_mss,speed_ms,0,blend_radius_m)
      movel([0.295795, -1.471305, -2.503183, -0.737901, 1.570796, 1.866592],accel_mss,speed_ms,0,blend_radius_m)
      movel([0.295324, -1.471069, -2.503381, -0.737938, 1.570796, 1.866120],accel_mss,speed_ms,0,blend_radius_m)
      movel([0.294866, -1.470819, -2.503591, -0.737978, 1.570796, 1.865662],accel_mss,speed_ms,0,blend_radius_m)
      movel([0.294417, -1.470559, -2.503810, -0.738020, 1.570796, 1.865213],accel_mss,speed_ms,0,blend_radius_m)
      movel([0.293983, -1.470285, -2.504041, -0.738063, 1.570796, 1.864779],accel_mss,speed_ms,0,blend_radius_m)
      movel([0.293559, -1.469998, -2.504282, -0.738109, 1.570796, 1.864355],accel_mss,speed_ms,0,blend_radius_m)
      movel([0.293149, -1.469699, -2.504533, -0.738157, 1.570796, 1.863946],accel_mss,speed_ms,0,blend_radius_m)
      movel([0.292750, -1.469387, -2.504794, -0.738208, 1.570796, 1.863546],accel_mss,speed_ms,0,blend_radius_m)
      movel([0.292420, -1.469107, -2.505029, -0.738253, 1.570796, 1.863216],accel_mss,speed_ms,0,blend_radius_m)
      movel([0.292102, -1.468815, -2.505274, -0.738300, 1.570796, 1.862898],accel_mss,speed_ms,0,blend_radius_m)
      movel([0.291798, -1.468512, -2.505528, -0.738349, 1.570796, 1.862595],accel_mss,speed_ms,0,blend_radius_m)
      movel([0.291509, -1.468196, -2.505792, -0.738401, 1.570796, 1.862305],accel_mss,speed_ms,0,blend_radius_m)
      movel([0.291236, -1.467869, -2.506065, -0.738454, 1.570796, 1.862032],accel_mss,speed_ms,0,blend_radius_m)
      movel([0.290975, -1.467530, -2.506349, -0.738510, 1.570796, 1.861771],accel_mss,speed_ms,0,blend_radius_m)
      movel([0.290729, -1.467182, -2.506640, -0.738567, 1.570796, 1.861525],accel_mss,speed_ms,0,blend_radius_m)
      movel([0.290549, -1.466896, -2.506879, -0.738614, 1.570796, 1.861346],accel_mss,speed_ms,0,blend_radius_m)
      movel([0.290383, -1.466602, -2.507124, -0.738663, 1.570796, 1.861180],accel_mss,speed_ms,0,blend_radius_m)
      movel([0.290233, -1.466298, -2.507378, -0.738713, 1.570796, 1.861029],accel_mss,speed_ms,0,blend_radius_m)
      movel([0.290095, -1.465985, -2.507638, -0.738765, 1.570796, 1.860892],accel_mss,speed_ms,0,blend_radius_m)
      movel([0.289976, -1.465664, -2.507906, -0.738819, 1.570796, 1.860772],accel_mss,speed_ms,0,blend_radius_m)
      movel([0.289869, -1.465335, -2.508180, -0.738874, 1.570796, 1.860665],accel_mss,speed_ms,0,blend_radius_m)
      movel([0.289780, -1.464997, -2.508461, -0.738931, 1.570796, 1.860576],accel_mss,speed_ms,0,blend_radius_m)
      movel([0.289703, -1.464652, -2.508748, -0.738989, 1.570796, 1.860500],accel_mss,speed_ms,0,blend_radius_m)
      movel([0.289650, -1.464346, -2.509003, -0.739040, 1.570796, 1.860447],accel_mss,speed_ms,0,blend_radius_m)
      movel([0.289607, -1.464035, -2.509261, -0.739093, 1.570796, 1.860404],accel_mss,speed_ms,0,blend_radius_m)
      movel([0.289577, -1.463719, -2.509523, -0.739147, 1.570796, 1.860373],accel_mss,speed_ms,0,blend_radius_m)
      movel([0.289553, -1.463400, -2.509787, -0.739201, 1.570796, 1.860349],accel_mss,speed_ms,0,blend_radius_m)
      movel([0.289545, -1.463117, -2.510022, -0.739249, 1.570796, 1.860342],accel_mss,speed_ms,0,blend_radius_m)
      movel([0.289550, -1.462829, -2.510261, -0.739299, 1.570796, 1.860346],accel_mss,speed_ms,0,blend_radius_m)
      movel([0.289571, -1.462536, -2.510504, -0.739349, 1.570796, 1.860367],accel_mss,speed_ms,0,blend_radius_m)
      movel([0.289603, -1.462241, -2.510748, -0.739400, 1.570796, 1.860399],accel_mss,speed_ms,0,blend_radius_m)
      movel([0.289651, -1.461918, -2.511015, -0.739456, 1.570796, 1.860447],accel_mss,speed_ms,0,blend_radius_m)
      movel([0.289714, -1.461594, -2.511283, -0.739512, 1.570796, 1.860510],accel_mss,speed_ms,0,blend_radius_m)
      movel([0.289789, -1.461266, -2.511554, -0.739569, 1.570796, 1.860585],accel_mss,speed_ms,0,blend_radius_m)
      movel([0.289875, -1.460938, -2.511825, -0.739626, 1.570796, 1.860671],accel_mss,speed_ms,0,blend_radius_m)
      movel([0.290046, -1.460366, -2.512297, -0.739726, 1.570796, 1.860843],accel_mss,speed_ms,0,blend_radius_m)
      movel([0.290229, -1.459793, -2.512770, -0.739827, 1.570796, 1.861025],accel_mss,speed_ms,0,blend_radius_m)
      movel([0.290425, -1.459218, -2.513243, -0.739928, 1.570796, 1.861221],accel_mss,speed_ms,0,blend_radius_m)
      movel([0.290736, -1.458366, -2.513944, -0.740080, 1.570796, 1.861532],accel_mss,speed_ms,0,blend_radius_m)
      movel([0.290875, -1.457998, -2.514246, -0.740145, 1.570796, 1.861671],accel_mss,speed_ms,0,blend_radius_m)
      movel([0.291019, -1.457630, -2.514548, -0.740211, 1.570796, 1.861815],accel_mss,speed_ms,0,blend_radius_m)
      movel([0.291273, -1.456998, -2.515066, -0.740325, 1.570796, 1.862069],accel_mss,speed_ms,0,blend_radius_m)
      movel([0.291289, -1.456967, -2.515091, -0.740331, 1.570796, 1.862085],accel_mss,speed_ms,0,blend_radius_m)
      movel([0.291312, -1.456936, -2.515117, -0.740336, 1.570796, 1.862109],accel_mss,speed_ms,0,blend_radius_m)
      movel([0.291342, -1.456910, -2.515138, -0.740341, 1.570796, 1.862138],accel_mss,speed_ms,0,blend_radius_m)
      movel([0.291377, -1.456889, -2.515155, -0.740345, 1.570796, 1.862173],accel_mss,speed_ms,0,blend_radius_m)
      movel([0.291414, -1.456878, -2.515164, -0.740347, 1.570796, 1.862211],accel_mss,speed_ms,0,blend_radius_m)
      movel([0.291449, -1.456877, -2.515165, -0.740347, 1.570796, 1.862245],accel_mss,speed_ms,0,blend_radius_m)
      movel([0.297738, -1.458121, -2.514145, -0.740123, 1.570796, 1.868535],accel_mss,speed_ms,0,blend_radius_m)
      movel([0.301205, -1.458828, -2.513564, -0.739997, 1.570796, 1.872001],accel_mss,speed_ms,0,blend_radius_m)
      movel([0.304655, -1.459556, -2.512965, -0.739868, 1.570796, 1.875452],accel_mss,speed_ms,0,blend_radius_m)
      movel([0.308729, -1.460440, -2.512236, -0.739713, 1.570796, 1.879525],accel_mss,speed_ms,0,blend_radius_m)
      movel([0.312786, -1.461345, -2.511489, -0.739555, 1.570796, 1.883582],accel_mss,speed_ms,0,blend_radius_m)
      movel([0.320904, -1.463225, -2.509933, -0.739231, 1.570796, 1.891700],accel_mss,speed_ms,0,blend_radius_m)
      movel([0.327823, -1.464893, -2.508548, -0.738948, 1.570796, 1.898620],accel_mss,speed_ms,0,blend_radius_m)
      movel([0.333854, -1.466399, -2.507293, -0.738697, 1.570796, 1.904650],accel_mss,speed_ms,0,blend_radius_m)
      movel([0.334793, -1.466645, -2.507088, -0.738656, 1.570796, 1.905589],accel_mss,speed_ms,0,blend_radius_m)
      movel([0.334922, -1.466689, -2.507051, -0.738648, 1.570796, 1.905718],accel_mss,speed_ms,0,blend_radius_m)
      movel([0.335045, -1.466737, -2.507011, -0.738640, 1.570796, 1.905842],accel_mss,speed_ms,0,blend_radius_m)
      speed_ms = 0.003
      movel([0.335045, -1.454665, -2.501542, -0.756183, 1.570796, 1.905842],accel_mss,speed_ms,0,blend_radius_m)
      speed_ms = 0.01
      movel([0.335045, -1.431374, -2.490212, -0.790803, 1.570796, 1.905842],accel_mss,speed_ms,0,blend_radius_m)
      movel([0.326327, -1.407583, -2.508609, -0.796197, 1.570796, 1.897124],accel_mss,speed_ms,0,blend_radius_m)
      movel([0.326327, -1.431348, -2.520227, -0.760815, 1.570796, 1.897124],accel_mss,speed_ms,0,blend_radius_m)
      speed_ms = 0.003
      movel([0.326327, -1.440572, -2.524449, -0.747368, 1.570796, 1.897124],accel_mss,speed_ms,0,blend_radius_m)
      speed_ms = 0.007
      movel([0.326287, -1.440595, -2.524431, -0.747363, 1.570796, 1.897083],accel_mss,speed_ms,0,blend_radius_m)
      movel([0.326246, -1.440611, -2.524418, -0.747360, 1.570796, 1.897043],accel_mss,speed_ms,0,blend_radius_m)
      movel([0.326206, -1.440616, -2.524414, -0.747359, 1.570796, 1.897002],accel_mss,speed_ms,0,blend_radius_m)
      movel([0.325298, -1.440616, -2.524414, -0.747359, 1.570796, 1.896095],accel_mss,speed_ms,0,blend_radius_m)
      movel([0.324773, -1.440614, -2.524416, -0.747360, 1.570796, 1.895569],accel_mss,speed_ms,0,blend_radius_m)
      movel([0.324253, -1.440603, -2.524424, -0.747362, 1.570796, 1.895049],accel_mss,speed_ms,0,blend_radius_m)
      movel([0.323648, -1.440587, -2.524437, -0.747365, 1.570796, 1.894444],accel_mss,speed_ms,0,blend_radius_m)
      movel([0.323042, -1.440566, -2.524453, -0.747369, 1.570796, 1.893839],accel_mss,speed_ms,0,blend_radius_m)
      movel([0.319909, -1.440454, -2.524543, -0.747392, 1.570796, 1.890706],accel_mss,speed_ms,0,blend_radius_m)
      movel([0.320130, -1.439955, -2.524939, -0.747495, 1.570796, 1.890926],accel_mss,speed_ms,0,blend_radius_m)
      movel([0.321415, -1.437070, -2.527224, -0.748095, 1.570796, 1.892212],accel_mss,speed_ms,0,blend_radius_m)
      movel([0.333621, -1.410066, -2.548005, -0.754318, 1.570796, 1.904417],accel_mss,speed_ms,0,blend_radius_m)
      movel([0.345787, -1.383626, -2.567307, -0.761456, 1.570796, 1.916583],accel_mss,speed_ms,0,blend_radius_m)
      movel([0.349559, -1.375532, -2.573014, -0.763843, 1.570796, 1.920355],accel_mss,speed_ms,0,blend_radius_m)
      movel([0.353527, -1.367044, -2.578898, -0.766447, 1.570796, 1.924323],accel_mss,speed_ms,0,blend_radius_m)
      movel([0.353557, -1.367015, -2.578918, -0.766456, 1.570796, 1.924353],accel_mss,speed_ms,0,blend_radius_m)
      movel([0.353600, -1.366987, -2.578937, -0.766465, 1.570796, 1.924396],accel_mss,speed_ms,0,blend_radius_m)
      movel([0.353645, -1.366966, -2.578951, -0.766472, 1.570796, 1.924441],accel_mss,speed_ms,0,blend_radius_m)
      movel([0.353705, -1.366949, -2.578963, -0.766477, 1.570796, 1.924502],accel_mss,speed_ms,0,blend_radius_m)
      movel([0.353761, -1.366943, -2.578967, -0.766479, 1.570796, 1.924558],accel_mss,speed_ms,0,blend_radius_m)
      movel([0.353825, -1.366942, -2.578968, -0.766479, 1.570796, 1.924621],accel_mss,speed_ms,0,blend_radius_m)
      movel([0.353884, -1.366947, -2.578964, -0.766478, 1.570796, 1.924680],accel_mss,speed_ms,0,blend_radius_m)
      movel([0.354117, -1.366971, -2.578948, -0.766470, 1.570796, 1.924914],accel_mss,speed_ms,0,blend_radius_m)
      movel([0.360561, -1.367263, -2.578747, -0.766379, 1.570796, 1.931357],accel_mss,speed_ms,0,blend_radius_m)
      movel([0.360888, -1.367285, -2.578732, -0.766372, 1.570796, 1.931684],accel_mss,speed_ms,0,blend_radius_m)
      movel([0.361210, -1.367315, -2.578711, -0.766363, 1.570796, 1.932007],accel_mss,speed_ms,0,blend_radius_m)
      movel([0.361527, -1.367352, -2.578686, -0.766351, 1.570796, 1.932324],accel_mss,speed_ms,0,blend_radius_m)
      movel([0.361688, -1.367382, -2.578665, -0.766342, 1.570796, 1.932485],accel_mss,speed_ms,0,blend_radius_m)
      movel([0.361843, -1.367421, -2.578638, -0.766330, 1.570796, 1.932640],accel_mss,speed_ms,0,blend_radius_m)
      movel([0.361990, -1.367470, -2.578605, -0.766314, 1.570796, 1.932786],accel_mss,speed_ms,0,blend_radius_m)
      movel([0.362028, -1.367493, -2.578589, -0.766307, 1.570796, 1.932824],accel_mss,speed_ms,0,blend_radius_m)
      movel([0.362057, -1.367525, -2.578567, -0.766297, 1.570796, 1.932854],accel_mss,speed_ms,0,blend_radius_m)
      movel([0.362071, -1.367567, -2.578538, -0.766284, 1.570796, 1.932867],accel_mss,speed_ms,0,blend_radius_m)
      movel([0.362070, -1.367617, -2.578503, -0.766268, 1.570796, 1.932867],accel_mss,speed_ms,0,blend_radius_m)
      movel([0.362054, -1.367670, -2.578467, -0.766252, 1.570796, 1.932851],accel_mss,speed_ms,0,blend_radius_m)
      movel([0.362015, -1.367754, -2.578409, -0.766226, 1.570796, 1.932811],accel_mss,speed_ms,0,blend_radius_m)
      movel([0.361958, -1.367839, -2.578351, -0.766199, 1.570796, 1.932755],accel_mss,speed_ms,0,blend_radius_m)
      movel([0.361922, -1.367879, -2.578323, -0.766187, 1.570796, 1.932718],accel_mss,speed_ms,0,blend_radius_m)
      movel([0.361878, -1.367913, -2.578300, -0.766176, 1.570796, 1.932674],accel_mss,speed_ms,0,blend_radius_m)
      movel([0.361830, -1.367941, -2.578281, -0.766167, 1.570796, 1.932626],accel_mss,speed_ms,0,blend_radius_m)
      movel([0.361765, -1.367965, -2.578264, -0.766160, 1.570796, 1.932561],accel_mss,speed_ms,0,blend_radius_m)
      movel([0.361702, -1.367982, -2.578253, -0.766155, 1.570796, 1.932498],accel_mss,speed_ms,0,blend_radius_m)
      movel([0.361640, -1.367992, -2.578246, -0.766151, 1.570796, 1.932436],accel_mss,speed_ms,0,blend_radius_m)
      movel([0.361486, -1.367998, -2.578241, -0.766150, 1.570796, 1.932282],accel_mss,speed_ms,0,blend_radius_m)
      movel([0.361334, -1.368000, -2.578240, -0.766149, 1.570796, 1.932130],accel_mss,speed_ms,0,blend_radius_m)
      movel([0.360745, -1.367984, -2.578251, -0.766154, 1.570796, 1.931541],accel_mss,speed_ms,0,blend_radius_m)
      movel([0.342925, -1.405247, -2.551599, -0.755542, 1.570796, 1.913721],accel_mss,speed_ms,0,blend_radius_m)
      movel([0.336455, -1.418983, -2.541263, -0.752142, 1.570796, 1.907251],accel_mss,speed_ms,0,blend_radius_m)
      movel([0.333782, -1.424688, -2.536889, -0.750813, 1.570796, 1.904578],accel_mss,speed_ms,0,blend_radius_m)
      movel([0.331134, -1.430345, -2.532502, -0.749542, 1.570796, 1.901931],accel_mss,speed_ms,0,blend_radius_m)
      movel([0.326420, -1.440460, -2.524538, -0.747391, 1.570796, 1.897216],accel_mss,speed_ms,0,blend_radius_m)
      movel([0.326396, -1.440502, -2.524505, -0.747383, 1.570796, 1.897193],accel_mss,speed_ms,0,blend_radius_m)
      movel([0.326366, -1.440538, -2.524476, -0.747375, 1.570796, 1.897162],accel_mss,speed_ms,0,blend_radius_m)
      movel([0.326327, -1.440572, -2.524449, -0.747368, 1.570796, 1.897124],accel_mss,speed_ms,0,blend_radius_m)
      speed_ms = 0.003
      movel([0.326327, -1.443685, -2.525839, -0.742864, 1.570796, 1.897124],accel_mss,speed_ms,0,blend_radius_m)
      speed_ms = 0.007
      movel([0.326287, -1.443708, -2.525821, -0.742860, 1.570796, 1.897083],accel_mss,speed_ms,0,blend_radius_m)
      movel([0.326246, -1.443724, -2.525808, -0.742857, 1.570796, 1.897043],accel_mss,speed_ms,0,blend_radius_m)
      movel([0.326206, -1.443728, -2.525805, -0.742856, 1.570796, 1.897002],accel_mss,speed_ms,0,blend_radius_m)
      movel([0.325298, -1.443729, -2.525804, -0.742856, 1.570796, 1.896095],accel_mss,speed_ms,0,blend_radius_m)
      movel([0.324773, -1.443726, -2.525806, -0.742856, 1.570796, 1.895569],accel_mss,speed_ms,0,blend_radius_m)
      movel([0.324253, -1.443716, -2.525815, -0.742858, 1.570796, 1.895049],accel_mss,speed_ms,0,blend_radius_m)
      movel([0.323648, -1.443700, -2.525827, -0.742861, 1.570796, 1.894444],accel_mss,speed_ms,0,blend_radius_m)
      movel([0.323042, -1.443679, -2.525844, -0.742866, 1.570796, 1.893839],accel_mss,speed_ms,0,blend_radius_m)
      movel([0.319909, -1.443567, -2.525934, -0.742888, 1.570796, 1.890706],accel_mss,speed_ms,0,blend_radius_m)
      movel([0.320130, -1.443070, -2.526331, -0.742988, 1.570796, 1.890926],accel_mss,speed_ms,0,blend_radius_m)
      movel([0.321415, -1.440193, -2.528620, -0.743575, 1.570796, 1.892212],accel_mss,speed_ms,0,blend_radius_m)
      movel([0.333621, -1.413266, -2.549444, -0.749678, 1.570796, 1.904417],accel_mss,speed_ms,0,blend_radius_m)
      movel([0.345787, -1.386900, -2.568789, -0.756700, 1.570796, 1.916583],accel_mss,speed_ms,0,blend_radius_m)
      movel([0.349559, -1.378827, -2.574509, -0.759053, 1.570796, 1.920355],accel_mss,speed_ms,0,blend_radius_m)
      movel([0.353527, -1.370362, -2.580407, -0.761620, 1.570796, 1.924323],accel_mss,speed_ms,0,blend_radius_m)
      movel([0.353557, -1.370333, -2.580427, -0.761629, 1.570796, 1.924353],accel_mss,speed_ms,0,blend_radius_m)
      movel([0.353600, -1.370306, -2.580446, -0.761638, 1.570796, 1.924396],accel_mss,speed_ms,0,blend_radius_m)
      movel([0.353645, -1.370285, -2.580460, -0.761644, 1.570796, 1.924441],accel_mss,speed_ms,0,blend_radius_m)
      movel([0.353705, -1.370267, -2.580472, -0.761650, 1.570796, 1.924502],accel_mss,speed_ms,0,blend_radius_m)
      movel([0.353761, -1.370262, -2.580476, -0.761651, 1.570796, 1.924558],accel_mss,speed_ms,0,blend_radius_m)
      movel([0.353825, -1.370260, -2.580477, -0.761652, 1.570796, 1.924621],accel_mss,speed_ms,0,blend_radius_m)
      movel([0.353884, -1.370265, -2.580473, -0.761650, 1.570796, 1.924680],accel_mss,speed_ms,0,blend_radius_m)
      movel([0.354117, -1.370289, -2.580457, -0.761643, 1.570796, 1.924914],accel_mss,speed_ms,0,blend_radius_m)
      movel([0.360561, -1.370580, -2.580256, -0.761553, 1.570796, 1.931357],accel_mss,speed_ms,0,blend_radius_m)
      movel([0.360888, -1.370603, -2.580240, -0.761546, 1.570796, 1.931684],accel_mss,speed_ms,0,blend_radius_m)
      movel([0.361210, -1.370632, -2.580220, -0.761537, 1.570796, 1.932007],accel_mss,speed_ms,0,blend_radius_m)
      movel([0.361527, -1.370669, -2.580194, -0.761525, 1.570796, 1.932324],accel_mss,speed_ms,0,blend_radius_m)
      movel([0.361688, -1.370699, -2.580174, -0.761516, 1.570796, 1.932485],accel_mss,speed_ms,0,blend_radius_m)
      movel([0.361843, -1.370738, -2.580147, -0.761504, 1.570796, 1.932640],accel_mss,speed_ms,0,blend_radius_m)
      movel([0.361990, -1.370787, -2.580113, -0.761489, 1.570796, 1.932786],accel_mss,speed_ms,0,blend_radius_m)
      movel([0.362028, -1.370810, -2.580097, -0.761482, 1.570796, 1.932824],accel_mss,speed_ms,0,blend_radius_m)
      movel([0.362057, -1.370842, -2.580075, -0.761472, 1.570796, 1.932854],accel_mss,speed_ms,0,blend_radius_m)
      movel([0.362071, -1.370884, -2.580046, -0.761459, 1.570796, 1.932867],accel_mss,speed_ms,0,blend_radius_m)
      movel([0.362070, -1.370934, -2.580011, -0.761444, 1.570796, 1.932867],accel_mss,speed_ms,0,blend_radius_m)
      movel([0.362054, -1.370987, -2.579975, -0.761427, 1.570796, 1.932851],accel_mss,speed_ms,0,blend_radius_m)
      movel([0.362015, -1.371070, -2.579917, -0.761402, 1.570796, 1.932811],accel_mss,speed_ms,0,blend_radius_m)
      movel([0.361958, -1.371155, -2.579859, -0.761376, 1.570796, 1.932755],accel_mss,speed_ms,0,blend_radius_m)
      movel([0.361922, -1.371195, -2.579831, -0.761363, 1.570796, 1.932718],accel_mss,speed_ms,0,blend_radius_m)
      movel([0.361878, -1.371229, -2.579807, -0.761353, 1.570796, 1.932674],accel_mss,speed_ms,0,blend_radius_m)
      movel([0.361830, -1.371257, -2.579788, -0.761344, 1.570796, 1.932626],accel_mss,speed_ms,0,blend_radius_m)
      movel([0.361765, -1.371281, -2.579772, -0.761337, 1.570796, 1.932561],accel_mss,speed_ms,0,blend_radius_m)
      movel([0.361702, -1.371297, -2.579760, -0.761332, 1.570796, 1.932498],accel_mss,speed_ms,0,blend_radius_m)
      movel([0.361640, -1.371308, -2.579753, -0.761328, 1.570796, 1.932436],accel_mss,speed_ms,0,blend_radius_m)
      movel([0.361486, -1.371314, -2.579749, -0.761327, 1.570796, 1.932282],accel_mss,speed_ms,0,blend_radius_m)
      movel([0.361334, -1.371315, -2.579748, -0.761326, 1.570796, 1.932130],accel_mss,speed_ms,0,blend_radius_m)
      movel([0.360745, -1.371300, -2.579758, -0.761331, 1.570796, 1.931541],accel_mss,speed_ms,0,blend_radius_m)
      movel([0.342925, -1.408461, -2.553046, -0.750882, 1.570796, 1.913721],accel_mss,speed_ms,0,blend_radius_m)
      movel([0.336455, -1.422159, -2.542688, -0.747542, 1.570796, 1.907251],accel_mss,speed_ms,0,blend_radius_m)
      movel([0.333782, -1.427846, -2.538304, -0.746238, 1.570796, 1.904578],accel_mss,speed_ms,0,blend_radius_m)
      movel([0.331134, -1.433487, -2.533909, -0.744993, 1.570796, 1.901931],accel_mss,speed_ms,0,blend_radius_m)
      movel([0.326420, -1.443573, -2.525929, -0.742887, 1.570796, 1.897216],accel_mss,speed_ms,0,blend_radius_m)
      movel([0.326396, -1.443615, -2.525896, -0.742879, 1.570796, 1.897193],accel_mss,speed_ms,0,blend_radius_m)
      movel([0.326366, -1.443651, -2.525867, -0.742871, 1.570796, 1.897162],accel_mss,speed_ms,0,blend_radius_m)
      movel([0.326327, -1.443685, -2.525839, -0.742864, 1.570796, 1.897124],accel_mss,speed_ms,0,blend_radius_m)
      speed_ms = 0.003
      movel([0.326327, -1.431348, -2.520227, -0.760815, 1.570796, 1.897124],accel_mss,speed_ms,0,blend_radius_m)
      speed_ms = 0.01
      movel([0.326327, -1.407583, -2.508609, -0.796197, 1.570796, 1.897124],accel_mss,speed_ms,0,blend_radius_m)
      movel([0.320882, -1.399907, -2.514372, -0.798110, 1.570796, 1.891678],accel_mss,speed_ms,0,blend_radius_m)
      movel([0.320882, -1.423822, -2.526083, -0.762483, 1.570796, 1.891678],accel_mss,speed_ms,0,blend_radius_m)
      speed_ms = 0.003
      movel([0.320882, -1.433110, -2.530340, -0.748939, 1.570796, 1.891678],accel_mss,speed_ms,0,blend_radius_m)
      speed_ms = 0.007
      movel([0.320788, -1.433140, -2.530316, -0.748932, 1.570796, 1.891585],accel_mss,speed_ms,0,blend_radius_m)
      movel([0.320696, -1.433160, -2.530301, -0.748928, 1.570796, 1.891492],accel_mss,speed_ms,0,blend_radius_m)
      movel([0.320606, -1.433174, -2.530290, -0.748925, 1.570796, 1.891402],accel_mss,speed_ms,0,blend_radius_m)
      movel([0.320280, -1.433201, -2.530268, -0.748919, 1.570796, 1.891076],accel_mss,speed_ms,0,blend_radius_m)
      movel([0.319953, -1.433225, -2.530250, -0.748914, 1.570796, 1.890749],accel_mss,speed_ms,0,blend_radius_m)
      movel([0.318880, -1.433294, -2.530196, -0.748899, 1.570796, 1.889676],accel_mss,speed_ms,0,blend_radius_m)
      movel([0.327715, -1.408533, -2.549152, -0.754704, 1.570796, 1.898511],accel_mss,speed_ms,0,blend_radius_m)
      movel([0.337071, -1.382780, -2.567908, -0.761701, 1.570796, 1.907867],accel_mss,speed_ms,0,blend_radius_m)
      movel([0.340564, -1.382538, -2.568080, -0.761771, 1.570796, 1.911360],accel_mss,speed_ms,0,blend_radius_m)
      movel([0.342544, -1.382415, -2.568167, -0.761807, 1.570796, 1.913340],accel_mss,speed_ms,0,blend_radius_m)
      movel([0.342990, -1.382396, -2.568180, -0.761812, 1.570796, 1.913786],accel_mss,speed_ms,0,blend_radius_m)
      movel([0.343429, -1.382396, -2.568180, -0.761812, 1.570796, 1.914226],accel_mss,speed_ms,0,blend_radius_m)
      movel([0.343585, -1.382404, -2.568175, -0.761810, 1.570796, 1.914381],accel_mss,speed_ms,0,blend_radius_m)
      movel([0.343736, -1.382418, -2.568165, -0.761806, 1.570796, 1.914532],accel_mss,speed_ms,0,blend_radius_m)
      movel([0.343881, -1.382442, -2.568148, -0.761799, 1.570796, 1.914678],accel_mss,speed_ms,0,blend_radius_m)
      movel([0.343922, -1.382461, -2.568134, -0.761793, 1.570796, 1.914719],accel_mss,speed_ms,0,blend_radius_m)
      movel([0.343950, -1.382493, -2.568112, -0.761784, 1.570796, 1.914746],accel_mss,speed_ms,0,blend_radius_m)
      movel([0.343960, -1.382538, -2.568080, -0.761771, 1.570796, 1.914757],accel_mss,speed_ms,0,blend_radius_m)
      movel([0.343948, -1.382590, -2.568043, -0.761756, 1.570796, 1.914744],accel_mss,speed_ms,0,blend_radius_m)
      movel([0.343903, -1.382705, -2.567961, -0.761723, 1.570796, 1.914699],accel_mss,speed_ms,0,blend_radius_m)
      movel([0.343853, -1.382819, -2.567881, -0.761690, 1.570796, 1.914650],accel_mss,speed_ms,0,blend_radius_m)
      movel([0.340662, -1.389756, -2.562923, -0.759710, 1.570796, 1.911458],accel_mss,speed_ms,0,blend_radius_m)
      movel([0.337163, -1.397387, -2.557389, -0.757613, 1.570796, 1.907959],accel_mss,speed_ms,0,blend_radius_m)
      movel([0.333104, -1.406279, -2.550832, -0.755277, 1.570796, 1.903901],accel_mss,speed_ms,0,blend_radius_m)
      movel([0.329072, -1.415158, -2.544170, -0.753061, 1.570796, 1.899869],accel_mss,speed_ms,0,blend_radius_m)
      movel([0.325605, -1.422835, -2.538315, -0.751239, 1.570796, 1.896401],accel_mss,speed_ms,0,blend_radius_m)
      movel([0.322683, -1.429331, -2.533291, -0.749766, 1.570796, 1.893480],accel_mss,speed_ms,0,blend_radius_m)
      movel([0.322096, -1.430634, -2.532276, -0.749479, 1.570796, 1.892892],accel_mss,speed_ms,0,blend_radius_m)
      movel([0.321129, -1.432851, -2.530543, -0.748995, 1.570796, 1.891925],accel_mss,speed_ms,0,blend_radius_m)
      movel([0.321091, -1.432921, -2.530488, -0.748980, 1.570796, 1.891888],accel_mss,speed_ms,0,blend_radius_m)
      movel([0.321042, -1.432991, -2.530433, -0.748965, 1.570796, 1.891838],accel_mss,speed_ms,0,blend_radius_m)
      movel([0.320997, -1.433039, -2.530396, -0.748954, 1.570796, 1.891793],accel_mss,speed_ms,0,blend_radius_m)
      movel([0.320943, -1.433079, -2.530364, -0.748946, 1.570796, 1.891739],accel_mss,speed_ms,0,blend_radius_m)
      movel([0.320882, -1.433110, -2.530340, -0.748939, 1.570796, 1.891678],accel_mss,speed_ms,0,blend_radius_m)
      speed_ms = 0.003
      movel([0.320882, -1.436244, -2.531743, -0.744402, 1.570796, 1.891678],accel_mss,speed_ms,0,blend_radius_m)
      speed_ms = 0.007
      movel([0.320788, -1.436275, -2.531719, -0.744395, 1.570796, 1.891585],accel_mss,speed_ms,0,blend_radius_m)
      movel([0.320696, -1.436295, -2.531703, -0.744391, 1.570796, 1.891492],accel_mss,speed_ms,0,blend_radius_m)
      movel([0.320606, -1.436309, -2.531692, -0.744388, 1.570796, 1.891402],accel_mss,speed_ms,0,blend_radius_m)
      movel([0.320280, -1.436336, -2.531671, -0.744383, 1.570796, 1.891076],accel_mss,speed_ms,0,blend_radius_m)
      movel([0.319953, -1.436359, -2.531653, -0.744378, 1.570796, 1.890749],accel_mss,speed_ms,0,blend_radius_m)
      movel([0.318880, -1.436428, -2.531598, -0.744363, 1.570796, 1.889676],accel_mss,speed_ms,0,blend_radius_m)
      movel([0.327715, -1.411738, -2.550593, -0.750057, 1.570796, 1.898511],accel_mss,speed_ms,0,blend_radius_m)
      movel([0.337071, -1.386056, -2.569392, -0.756942, 1.570796, 1.907867],accel_mss,speed_ms,0,blend_radius_m)
      movel([0.340564, -1.385815, -2.569563, -0.757011, 1.570796, 1.911360],accel_mss,speed_ms,0,blend_radius_m)
      movel([0.342544, -1.385692, -2.569651, -0.757046, 1.570796, 1.913340],accel_mss,speed_ms,0,blend_radius_m)
      movel([0.342990, -1.385673, -2.569664, -0.757052, 1.570796, 1.913786],accel_mss,speed_ms,0,blend_radius_m)
      movel([0.343429, -1.385673, -2.569664, -0.757052, 1.570796, 1.914226],accel_mss,speed_ms,0,blend_radius_m)
      movel([0.343585, -1.385681, -2.569659, -0.757049, 1.570796, 1.914381],accel_mss,speed_ms,0,blend_radius_m)
      movel([0.343736, -1.385695, -2.569648, -0.757045, 1.570796, 1.914532],accel_mss,speed_ms,0,blend_radius_m)
      movel([0.343881, -1.385719, -2.569632, -0.757038, 1.570796, 1.914678],accel_mss,speed_ms,0,blend_radius_m)
      movel([0.343922, -1.385738, -2.569618, -0.757033, 1.570796, 1.914719],accel_mss,speed_ms,0,blend_radius_m)
      movel([0.343950, -1.385770, -2.569595, -0.757024, 1.570796, 1.914746],accel_mss,speed_ms,0,blend_radius_m)
      movel([0.343960, -1.385815, -2.569563, -0.757011, 1.570796, 1.914757],accel_mss,speed_ms,0,blend_radius_m)
      movel([0.343948, -1.385866, -2.569526, -0.756996, 1.570796, 1.914744],accel_mss,speed_ms,0,blend_radius_m)
      movel([0.343903, -1.385982, -2.569444, -0.756963, 1.570796, 1.914699],accel_mss,speed_ms,0,blend_radius_m)
      movel([0.343853, -1.386095, -2.569364, -0.756931, 1.570796, 1.914650],accel_mss,speed_ms,0,blend_radius_m)
      movel([0.340662, -1.393013, -2.564394, -0.754981, 1.570796, 1.911458],accel_mss,speed_ms,0,blend_radius_m)
      movel([0.337163, -1.400623, -2.558848, -0.752918, 1.570796, 1.907959],accel_mss,speed_ms,0,blend_radius_m)
      movel([0.333104, -1.409491, -2.552277, -0.750621, 1.570796, 1.903901],accel_mss,speed_ms,0,blend_radius_m)
      movel([0.329072, -1.418344, -2.545600, -0.748444, 1.570796, 1.899869],accel_mss,speed_ms,0,blend_radius_m)
      movel([0.325605, -1.426000, -2.539733, -0.746656, 1.570796, 1.896401],accel_mss,speed_ms,0,blend_radius_m)
      movel([0.322683, -1.432477, -2.534700, -0.745213, 1.570796, 1.893480],accel_mss,speed_ms,0,blend_radius_m)
      movel([0.322096, -1.433776, -2.533683, -0.744931, 1.570796, 1.892892],accel_mss,speed_ms,0,blend_radius_m)
      movel([0.321129, -1.435986, -2.531946, -0.744457, 1.570796, 1.891925],accel_mss,speed_ms,0,blend_radius_m)
      movel([0.321091, -1.436056, -2.531891, -0.744442, 1.570796, 1.891888],accel_mss,speed_ms,0,blend_radius_m)
      movel([0.321042, -1.436126, -2.531836, -0.744427, 1.570796, 1.891838],accel_mss,speed_ms,0,blend_radius_m)
      movel([0.320997, -1.436174, -2.531798, -0.744417, 1.570796, 1.891793],accel_mss,speed_ms,0,blend_radius_m)
      movel([0.320943, -1.436214, -2.531767, -0.744408, 1.570796, 1.891739],accel_mss,speed_ms,0,blend_radius_m)
      movel([0.320882, -1.436244, -2.531743, -0.744402, 1.570796, 1.891678],accel_mss,speed_ms,0,blend_radius_m)
      speed_ms = 0.003
      movel([0.320882, -1.423822, -2.526083, -0.762483, 1.570796, 1.891678],accel_mss,speed_ms,0,blend_radius_m)
      speed_ms = 0.01
      movel([0.320882, -1.399907, -2.514372, -0.798110, 1.570796, 1.891678],accel_mss,speed_ms,0,blend_radius_m)
      movel([0.344723, -1.324283, -2.566799, -0.821307, 1.570796, 1.915519],accel_mss,speed_ms,0,blend_radius_m)
